KUKA KRL program: MyProgram_096().src

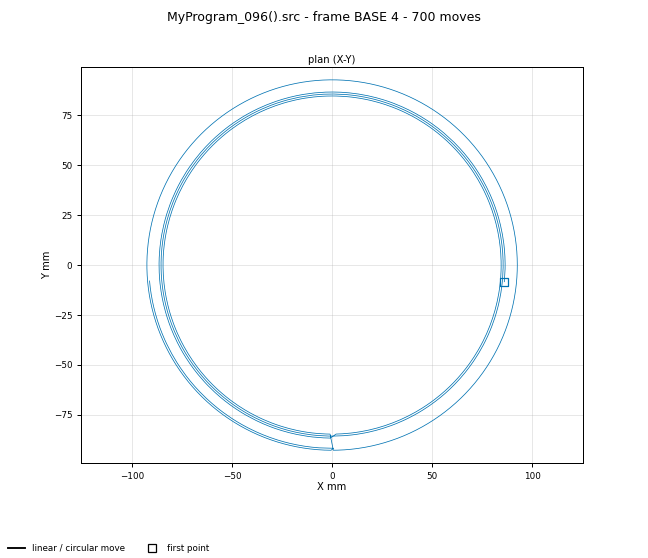
[picture p0: tool path of MyProgram_096().src in frame BASE 4, 700 of 700 moves have a stored position in this frame; points joined in program order, loops and branches not executed]
&ACCESS RVP
&REL 1
&PARAM TEMPLATE = C:\KRC\Roboter\Template\vorgabe
&PARAM EDITMASK = *
DEF MyProgram_096()
; ---- Setting reference (Base) ----
$BASE = BASE_DATA[4]

; --------------------------
; ---- Setting tool (TCP) ----
$TOOL = TOOL_DATA[3]
; --------------------------

$VEL.CP = VEL_APROX_PRINT
Startdeposition()
$VEL.CP = VEL_PRINT
LIN {X 86.1652,Y -8.3322,Z 89,A -10.037,B 24.913,C -2.1541,E1 25.1592,E2 454.8857} C_DIS
LIN {X 86.5449,Y -1.9567,Z 89,A -6.1016,B 24.9127,C -2.1574,E1 25.1598,E2 450.966} C_DIS
LIN {X 86.5649,Y 0.564,Z 89,A -3.5482,B 24.9097,C -2.1938,E1 25.1598,E2 448.3417} C_DIS
LIN {X 86.4537,Y 4.4277,Z 89,A -1.0805,B 24.9093,C -2.1987,E1 25.1594,E2 445.8771} C_DIS
LIN {X 86.1959,Y 7.9991,Z 89,A 0.4802,B 24.911,C -2.1778,E1 25.159,E2 444.3749} C_DIS
LIN {X 85.8962,Y 10.7562,Z 89,A 3.3475,B 24.9076,C -2.2199,E1 25.158,E2 441.4254} C_DIS
LIN {X 85.2355,Y 15.1219,Z 89,A 5.3712,B 24.9094,C -2.1974,E1 25.1571,E2 439.4666} C_DIS
LIN {X 84.2333,Y 19.9676,Z 89,A 8.7324,B 24.9083,C -2.2104,E1 25.1551,E2 436.0942} C_DIS
LIN {X 83.3839,Y 23.2585,Z 89,A 11.371,B 24.9066,C -2.2309,E1 25.1531,E2 433.4224} C_DIS
LIN {X 82.4594,Y 26.3489,Z 89,A 13.082,B 24.9073,C -2.2224,E1 25.1517,E2 431.7411} C_DIS
LIN {X 81.4082,Y 29.4361,Z 89,A 15.0667,B 24.9073,C -2.2228,E1 25.1499,E2 429.7667} C_DIS
LIN {X 80.3466,Y 32.2233,Z 89,A 17.2208,B 24.9063,C -2.2347,E1 25.1476,E2 427.5963} C_DIS
LIN {X 79.0048,Y 35.3836,Z 89,A 19.357,B 24.9062,C -2.2365,E1 25.1453,E2 425.4676} C_DIS
LIN {X 77.227,Y 39.1127,Z 89,A 22.0396,B 24.9057,C -2.2423,E1 25.142,E2 422.7857} C_DIS
LIN {X 75.0008,Y 43.2274,Z 89,A 24.8005,B 24.9059,C -2.2392,E1 25.1383,E2 420.0465} C_DIS
LIN {X 73.7426,Y 45.3426,Z 89,A 26.77,B 24.9046,C -2.2551,E1 25.1354,E2 418.0496} C_DIS
LIN {X 71.7448,Y 48.4398,Z 89,A 29.0057,B 24.9046,C -2.2544,E1 25.132,E2 415.8267} C_DIS
LIN {X 70.1596,Y 50.7113,Z 89,A 31.6144,B 24.902,C -2.2854,E1 25.1277,E2 413.1572} C_DIS
LIN {X 68.0698,Y 53.4816,Z 89,A 33.2305,B 24.9035,C -2.2677,E1 25.125,E2 411.5907} C_DIS
LIN {X 66.2061,Y 55.7736,Z 89,A 35.314,B 24.9028,C -2.2766,E1 25.1212,E2 409.4958} C_DIS
LIN {X 64.0318,Y 58.2561,Z 89,A 38.2857,B 24.9,C -2.3083,E1 25.1156,E2 406.4622} C_DIS
LIN {X 60.9971,Y 61.4257,Z 89,A 40.2743,B 24.9022,C -2.2834,E1 25.1118,E2 404.541} C_DIS
LIN {X 56.0568,Y 65.9649,Z 89,A 44.1821,B 24.9029,C -2.2744,E1 25.1038,E2 400.6702} C_DIS
LIN {X 53.2501,Y 68.2526,Z 89,A 47.0391,B 24.9013,C -2.2941,E1 25.0975,E2 397.7774} C_DIS
LIN {X 50.041,Y 70.6378,Z 89,A 49.6019,B 24.9011,C -2.2959,E1 25.0917,E2 395.2194} C_DIS
LIN {X 47.7464,Y 72.2081,Z 89,A 51.972,B 24.8993,C -2.3165,E1 25.0861,E2 392.8085} C_DIS
LIN {X 44.2677,Y 74.3919,Z 89,A 54.2125,B 24.9003,C -2.3047,E1 25.0809,E2 390.603} C_DIS
LIN {X 41.8224,Y 75.7944,Z 89,A 56.1926,B 24.8998,C -2.3111,E1 25.076,E2 388.6136} C_DIS
LIN {X 38.5837,Y 77.4922,Z 89,A 58.4027,B 24.9001,C -2.3073,E1 25.0706,E2 386.4186} C_DIS
LIN {X 34.9888,Y 79.1814,Z 89,A 61.2752,B 24.8992,C -2.3183,E1 25.0633,E2 383.5273} C_DIS
LIN {X 30.7564,Y 80.9183,Z 89,A 63.8229,B 24.9002,C -2.3058,E1 25.0568,E2 381.0151} C_DIS
LIN {X 28.2145,Y 81.8406,Z 89,A 65.9642,B 24.8991,C -2.3187,E1 25.051,E2 378.8475} C_DIS
LIN {X 25.6479,Y 82.6795,Z 89,A 67.7739,B 24.8989,C -2.3208,E1 25.0462,E2 377.0361} C_DIS
LIN {X 22.2469,Y 83.6595,Z 89,A 70.3552,B 24.8981,C -2.33,E1 25.0392,E2 374.4372} C_DIS
LIN {X 18.0288,Y 84.6691,Z 89,A 72.9776,B 24.8987,C -2.3235,E1 25.0321,E2 371.8337} C_DIS
LIN {X 13.1799,Y 85.557,Z 89,A 77.2175,B 24.8959,C -2.3559,E1 25.0203,E2 367.5214} C_DIS
LIN {X 8.4606,Y 86.1533,Z 89,A 79.4585,B 24.8984,C -2.3274,E1 25.0142,E2 365.3495} C_DIS
LIN {X 4.3743,Y 86.4555,Z 89,A 82.1881,B 24.8984,C -2.328,E1 25.0066,E2 362.6195} C_DIS
LIN {X 0.4649,Y 86.565,Z 89,A 84.9734,B 24.8978,C -2.3338,E1 24.9988,E2 359.821} C_DIS
LIN {X -3.1987,Y 86.5087,Z 89,A 88.381,B 24.8951,C -2.3638,E1 24.9891,E2 356.3412} C_DIS
LIN {X -8.7789,Y 86.1203,Z 89,A 90.702,B 24.8991,C -2.319,E1 24.9829,E2 354.1257} C_DIS
LIN {X -14.3867,Y 85.3625,Z 89,A 94.3706,B 24.8995,C -2.3142,E1 24.9728,E2 350.4655} C_DIS
LIN {X -17.7226,Y 84.7333,Z 89,A 97.0609,B 24.8985,C -2.3259,E1 24.9654,E2 347.7444} C_DIS
LIN {X -21.2707,Y 83.9126,Z 89,A 99.7429,B 24.898,C -2.3319,E1 24.958,E2 345.0444} C_DIS
LIN {X -24.8815,Y 82.9138,Z 89,A 101.8095,B 24.8993,C -2.3166,E1 24.9526,E2 343.0107} C_DIS
LIN {X -28.1429,Y 81.8655,Z 89,A 104.0096,B 24.8997,C -2.3119,E1 24.9468,E2 340.8178} C_DIS
LIN {X -32.7128,Y 80.1473,Z 89,A 107.0659,B 24.9005,C -2.3023,E1 24.9389,E2 337.7777} C_DIS
LIN {X -36.9162,Y 78.3013,Z 89,A 110.2494,B 24.9005,C -2.3021,E1 24.9307,E2 334.5871} C_DIS
LIN {X -39.8368,Y 76.8569,Z 89,A 112.4132,B 24.9009,C -2.2988,E1 24.9253,E2 332.4253} C_DIS
LIN {X -42.6915,Y 75.3087,Z 89,A 114.5747,B 24.9011,C -2.2955,E1 24.9201,E2 330.2655} C_DIS
LIN {X -44.87,Y 74.0298,Z 89,A 116.3495,B 24.9011,C -2.2955,E1 24.9158,E2 328.4852} C_DIS
LIN {X -49.0838,Y 71.3068,Z 89,A 119.6977,B 24.9016,C -2.2899,E1 24.908,E2 325.1394} C_DIS
LIN {X -51.7362,Y 69.406,Z 89,A 122.1888,B 24.9012,C -2.2952,E1 24.9024,E2 322.6269} C_DIS
LIN {X -54.4997,Y 67.257,Z 89,A 124.5303,B 24.9015,C -2.2909,E1 24.8973,E2 320.2868} C_DIS
LIN {X -58.1437,Y 64.135,Z 89,A 127.8803,B 24.9017,C -2.2888,E1 24.8903,E2 316.9286} C_DIS
LIN {X -60.4941,Y 61.9199,Z 89,A 129.6741,B 24.903,C -2.2737,E1 24.8867,E2 315.1632} C_DIS
LIN {X -63.2937,Y 59.0571,Z 89,A 132.285,B 24.9037,C -2.2661,E1 24.8817,E2 312.5592} C_DIS
LIN {X -65.8738,Y 56.1637,Z 89,A 135.6513,B 24.9022,C -2.2827,E1 24.8755,E2 309.1378} C_DIS
LIN {X -68.7539,Y 52.5995,Z 89,A 137.668,B 24.9054,C -2.2454,E1 24.8722,E2 307.2008} C_DIS
LIN {X -71.5133,Y 48.7816,Z 89,A 140.6821,B 24.9064,C -2.2339,E1 24.8673,E2 304.1992} C_DIS
LIN {X -72.8089,Y 46.825,Z 89,A 142.4997,B 24.9061,C -2.2371,E1 24.8645,E2 302.3648} C_DIS
LIN {X -75.3983,Y 42.5318,Z 89,A 145.8903,B 24.9067,C -2.2297,E1 24.8597,E2 298.9745} C_DIS
LIN {X -76.9384,Y 39.6775,Z 89,A 147.9529,B 24.9075,C -2.221,E1 24.857,E2 296.9215} C_DIS
LIN {X -78.2041,Y 37.1214,Z 89,A 149.991,B 24.9075,C -2.2197,E1 24.8545,E2 294.8756} C_DIS
LIN {X -80.0414,Y 32.9731,Z 89,A 152.6386,B 24.9092,C -2.2006,E1 24.8516,E2 292.2589} C_DIS
LIN {X -80.9706,Y 30.6182,Z 89,A 154.878,B 24.9083,C -2.2114,E1 24.8494,E2 289.9811} C_DIS
LIN {X -82.6055,Y 25.8867,Z 89,A 158.1523,B 24.9092,C -2.2001,E1 24.8465,E2 286.7152} C_DIS
LIN {X -83.441,Y 23.0556,Z 89,A 159.9044,B 24.9102,C -2.1882,E1 24.8452,E2 284.9813} C_DIS
LIN {X -84.156,Y 20.2864,Z 89,A 161.7857,B 24.9107,C -2.1819,E1 24.8439,E2 283.1039} C_DIS
LIN {X -85.1399,Y 15.6532,Z 89,A 165.0153,B 24.9113,C -2.1746,E1 24.8421,E2 279.8727} C_DIS
LIN {X -85.6777,Y 12.3726,Z 89,A 167.8753,B 24.9103,C -2.1863,E1 24.841,E2 276.9677} C_DIS
LIN {X -86.149,Y 8.5042,Z 89,A 169.6403,B 24.9129,C -2.155,E1 24.8405,E2 275.2669} C_DIS
LIN {X -86.4853,Y 3.7439,Z 89,A 172.8591,B 24.9136,C -2.1466,E1 24.8399,E2 272.0489} C_DIS
LIN {X -86.5642,Y 0.6968,Z 89,A 175.0036,B 24.9138,C -2.1437,E1 24.8398,E2 269.8984} C_DIS
LIN {X -86.4823,Y -3.8138,Z 89,A 178.5276,B 24.9133,C -2.1494,E1 24.8401,E2 266.3394} C_DIS
LIN {X -86.2728,Y -7.126,Z 89,A 179.9255,B 24.9157,C -2.1199,E1 24.8404,E2 265.0037} C_DIS
LIN {X -86.056,Y -9.3927,Z 89,A -177.5698,B 24.9138,C -2.1434,E1 24.8412,E2 262.4278} C_DIS
LIN {X -85.5563,Y -13.185,Z 89,A -175.8758,B 24.9164,C -2.1117,E1 24.8418,E2 260.7995} C_DIS
LIN {X -84.9399,Y -16.705,Z 89,A -173.2886,B 24.9164,C -2.1106,E1 24.8431,E2 258.1996} C_DIS
LIN {X -84.2882,Y -19.7303,Z 89,A -171.2652,B 24.917,C -2.1036,E1 24.8444,E2 256.1809} C_DIS
LIN {X -83.3415,Y -23.4082,Z 89,A -169.0394,B 24.9183,C -2.0878,E1 24.846,E2 253.9799} C_DIS
LIN {X -82.6319,Y -25.8014,Z 89,A -167.0637,B 24.9179,C -2.092,E1 24.8476,E2 251.9827} C_DIS
LIN {X -81.5331,Y -29.0907,Z 89,A -164.6138,B 24.9181,C -2.0897,E1 24.8498,E2 249.5246} C_DIS
LIN {X -80.5182,Y -31.7893,Z 89,A -162.9315,B 24.919,C -2.0777,E1 24.8515,E2 247.8614} C_DIS
LIN {X -79.1289,Y -35.1047,Z 89,A -160.0378,B 24.9184,C -2.0857,E1 24.8548,E2 244.9325} C_DIS
LIN {X -77.4475,Y -38.6738,Z 89,A -157.6886,B 24.9196,C -2.0709,E1 24.8576,E2 242.606} C_DIS
LIN {X -75.9339,Y -41.5677,Z 89,A -155.686,B 24.9204,C -2.0604,E1 24.8602,E2 240.6178} C_DIS
LIN {X -74.4678,Y -44.1393,Z 89,A -153.6152,B 24.9205,C -2.0585,E1 24.8632,E2 238.5409} C_DIS
LIN {X -73.1265,Y -46.3303,Z 89,A -152.1316,B 24.9214,C -2.0478,E1 24.8653,E2 237.0753} C_DIS
LIN {X -71.2162,Y -49.2139,Z 89,A -149.0869,B 24.9201,C -2.064,E1 24.8702,E2 233.9767} C_DIS
LIN {X -69.1788,Y -52.0385,Z 89,A -147.1357,B 24.9213,C -2.0481,E1 24.8734,E2 232.0542} C_DIS
LIN {X -67.1011,Y -54.692,Z 89,A -145.069,B 24.9221,C -2.038,E1 24.877,E2 230.0018} C_DIS
LIN {X -63.8641,Y -58.4389,Z 89,A -142.2392,B 24.9237,C -2.0175,E1 24.8822,E2 227.2081} C_DIS
LIN {X -62.2823,Y -60.1219,Z 89,A -140.3571,B 24.9231,C -2.0245,E1 24.8858,E2 225.3011} C_DIS
LIN {X -58.6037,Y -63.7129,Z 89,A -136.8514,B 24.9234,C -2.0206,E1 24.8929,E2 221.7902} C_DIS
LIN {X -56.0418,Y -65.9776,Z 89,A -134.6035,B 24.9238,C -2.0158,E1 24.8976,E2 219.5451} C_DIS
LIN {X -53.545,Y -68.0196,Z 89,A -132.3743,B 24.9238,C -2.0147,E1 24.9025,E2 217.3101} C_DIS
LIN {X -50.9969,Y -69.9504,Z 89,A -129.8993,B 24.9233,C -2.0219,E1 24.9081,E2 214.8092} C_DIS
LIN {X -48.1446,Y -71.9447,Z 89,A -127.8708,B 24.9243,C -2.0098,E1 24.9128,E2 212.8027} C_DIS
LIN {X -45.3206,Y -73.756,Z 89,A -125.9165,B 24.9251,C -1.9984,E1 24.9173,E2 210.8692} C_DIS
LIN {X -43.0007,Y -75.1311,Z 89,A -123.765,B 24.9245,C -2.007,E1 24.9226,E2 208.6908} C_DIS
LIN {X -37.8884,Y -77.8356,Z 89,A -120.3477,B 24.9258,C -1.9896,E1 24.931,E2 205.3056} C_DIS
LIN {X -34.2947,Y -79.4839,Z 89,A -117.631,B 24.9258,C -1.9898,E1 24.9379,E2 202.5819} C_DIS
LIN {X -31.1627,Y -80.7643,Z 89,A -115.3064,B 24.9258,C -1.9902,E1 24.944,E2 200.2512} C_DIS
LIN {X -28.6047,Y -81.7037,Z 89,A -113.5823,B 24.926,C -1.9862,E1 24.9485,E2 198.5332} C_DIS
LIN {X -25.2724,Y -82.7959,Z 89,A -110.8821,B 24.9253,C -1.9963,E1 24.9558,E2 195.8044} C_DIS
LIN {X -21.5951,Y -83.8294,Z 89,A -108.5996,B 24.926,C -1.9871,E1 24.9619,E2 193.5403} C_DIS
LIN {X -17.6457,Y -84.7486,Z 89,A -106.0736,B 24.9264,C -1.9809,E1 24.9687,E2 191.0258} C_DIS
LIN {X -12.0537,Y -85.723,Z 89,A -102.4921,B 24.9269,C -1.9741,E1 24.9786,E2 187.4568} C_DIS
LIN {X -9.5862,Y -86.0352,Z 89,A -100.3696,B 24.9258,C -1.9889,E1 24.9845,E2 185.2978} C_DIS
LIN {X -4.2582,Y -86.4608,Z 89,A -96.8864,B 24.926,C -1.9873,E1 24.9942,E2 181.8172} C_DIS
LIN {X -0.9571,Y -86.562,Z 89,A -94.6458,B 24.9258,C -1.9894,E1 25.0005,E2 179.5716} C_DIS
LIN {X -0.9571,Y -86.562,Z 89,A -94.6458,B 24.9258,C -1.9894,E1 25.0005,E2 179.5716} C_DIS
Enddeposition()
LIN {X 0.5384,Y -85.5676,Z 89,A -92.9762,B 24.9228,C -2.0285,E1 25.0055,E2 177.8093} C_DIS
Startdeposition()
$VEL.CP = VEL_PRINT
LIN {X -1.8149,Y -85.5541,Z 89,A -96.7949,B 24.9282,C -1.9573,E1 24.9943,E2 181.7968} C_DIS
LIN {X -7.3834,Y -85.2553,Z 89,A -99.9511,B 24.9269,C -1.975,E1 24.9856,E2 184.9121} C_DIS
LIN {X -10.1639,Y -84.9675,Z 89,A -101.8253,B 24.9269,C -1.9752,E1 24.9804,E2 186.787} C_DIS
LIN {X -14.2461,Y -84.379,Z 89,A -104.8301,B 24.9274,C -1.9684,E1 24.9721,E2 189.8105} C_DIS
LIN {X -18.2268,Y -83.6094,Z 89,A -107.4223,B 24.927,C -1.9733,E1 24.965,E2 192.3942} C_DIS
LIN {X -21.0814,Y -82.9359,Z 89,A -109.4344,B 24.927,C -1.9729,E1 24.9595,E2 194.41} C_DIS
LIN {X -23.2275,Y -82.3604,Z 89,A -110.8461,B 24.9268,C -1.9761,E1 24.9557,E2 195.8162} C_DIS
LIN {X -25.9725,Y -81.5373,Z 89,A -112.9249,B 24.927,C -1.9727,E1 24.9502,E2 197.9068} C_DIS
LIN {X -29.1962,Y -80.4385,Z 89,A -115.1571,B 24.9268,C -1.976,E1 24.9443,E2 200.1353} C_DIS
LIN {X -32.3957,Y -79.2041,Z 89,A -117.498,B 24.9268,C -1.9769,E1 24.9382,E2 202.4792} C_DIS
LIN {X -34.7519,Y -78.1996,Z 89,A -119.2917,B 24.9268,C -1.9764,E1 24.9336,E2 204.2784} C_DIS
LIN {X -38.4653,Y -76.4417,Z 89,A -121.9779,B 24.9264,C -1.9816,E1 24.9269,E2 206.9593} C_DIS
LIN {X -40.873,Y -75.1807,Z 89,A -123.6243,B 24.9258,C -1.9891,E1 24.9228,E2 208.5924} C_DIS
LIN {X -43.3867,Y -73.7589,Z 89,A -125.7047,B 24.9259,C -1.9875,E1 24.9178,E2 210.6828} C_DIS
LIN {X -46.2938,Y -71.9696,Z 89,A -128.0158,B 24.9257,C -1.9902,E1 24.9123,E2 212.9948} C_DIS
LIN {X -48.9738,Y -70.1736,Z 89,A -130.2026,B 24.9255,C -1.9929,E1 24.9073,E2 215.1825} C_DIS
LIN {X -51.5458,Y -68.3067,Z 89,A -132.2676,B 24.9251,C -1.9984,E1 24.9027,E2 217.2417} C_DIS
LIN {X -54.0811,Y -66.3178,Z 89,A -134.508,B 24.9251,C -1.9999,E1 24.8978,E2 219.4869} C_DIS
LIN {X -56.6656,Y -64.1249,Z 89,A -136.8256,B 24.9248,C -2.0029,E1 24.8929,E2 221.8065} C_DIS
LIN {X -58.5379,Y -62.4186,Z 89,A -138.4467,B 24.9244,C -2.0085,E1 24.8896,E2 223.4209} C_DIS
LIN {X -60.8702,Y -60.1462,Z 89,A -140.5817,B 24.9239,C -2.0143,E1 24.8853,E2 225.551} C_DIS
LIN {X -63.0112,Y -57.8994,Z 89,A -142.5919,B 24.9234,C -2.0208,E1 24.8815,E2 227.5546} C_DIS
LIN {X -64.8576,Y -55.8249,Z 89,A -144.6641,B 24.9236,C -2.0189,E1 24.8777,E2 229.6406} C_DIS
LIN {X -67.051,Y -53.1689,Z 89,A -146.7937,B 24.9228,C -2.0293,E1 24.8739,E2 231.7552} C_DIS
LIN {X -69.5729,Y -49.8234,Z 89,A -150.249,B 24.9236,C -2.018,E1 24.8682,E2 235.2544} C_DIS
LIN {X -71.3942,Y -47.1765,Z 89,A -151.5228,B 24.9214,C -2.048,E1 24.8663,E2 236.4629} C_DIS
LIN {X -73.247,Y -44.2456,Z 89,A -154.2983,B 24.9219,C -2.0412,E1 24.8621,E2 239.2686} C_DIS
LIN {X -74.9459,Y -41.3047,Z 89,A -156.6234,B 24.9215,C -2.0459,E1 24.8589,E2 241.5949} C_DIS
LIN {X -76.6041,Y -38.1389,Z 89,A -158.5908,B 24.9201,C -2.0643,E1 24.8565,E2 243.5288} C_DIS
LIN {X -78.9168,Y -33.0893,Z 89,A -162.522,B 24.9197,C -2.0688,E1 24.8519,E2 247.4707} C_DIS
LIN {X -80.3338,Y -29.4832,Z 89,A -165.2714,B 24.9195,C -2.0721,E1 24.8492,E2 250.2278} C_DIS
LIN {X -81.439,Y -26.2762,Z 89,A -167.6499,B 24.9192,C -2.0759,E1 24.8471,E2 252.611} C_DIS
LIN {X -82.4274,Y -22.991,Z 89,A -169.952,B 24.9187,C -2.0826,E1 24.8453,E2 254.9102} C_DIS
LIN {X -83.2905,Y -19.6361,Z 89,A -171.9622,B 24.9174,C -2.0982,E1 24.8439,E2 256.895} C_DIS
LIN {X -83.8501,Y -17.0858,Z 89,A -174.0038,B 24.9176,C -2.0955,E1 24.8427,E2 258.9549} C_DIS
LIN {X -84.4897,Y -13.5829,Z 89,A -176.2039,B 24.9167,C -2.1079,E1 24.8417,E2 261.1385} C_DIS
LIN {X -84.8798,Y -10.8714,Z 89,A -178.1199,B 24.9164,C -2.1115,E1 24.8409,E2 263.0575} C_DIS
LIN {X -85.2436,Y -7.5095,Z 89,A 179.5778,B 24.9159,C -2.1176,E1 24.8403,E2 265.359} C_DIS
LIN {X -85.4548,Y -4.5016,Z 89,A 177.5208,B 24.9155,C -2.1229,E1 24.8399,E2 267.4156} C_DIS
LIN {X -85.5573,Y -1.6423,Z 89,A 175.57,B 24.9151,C -2.1281,E1 24.8398,E2 269.3659} C_DIS
LIN {X -85.5639,Y 1.2851,Z 89,A 173.5749,B 24.9146,C -2.1334,E1 24.8398,E2 271.3603} C_DIS
LIN {X -85.4292,Y 4.965,Z 89,A 170.9832,B 24.9143,C -2.1379,E1 24.8402,E2 273.9569} C_DIS
LIN {X -85.1495,Y 8.5125,Z 89,A 168.4041,B 24.9141,C -2.1401,E1 24.8408,E2 276.546} C_DIS
LIN {X -84.6897,Y 12.2655,Z 89,A 166.2108,B 24.9127,C -2.1574,E1 24.8416,E2 278.7112} C_DIS
LIN {X -84.2353,Y 15.0718,Z 89,A 164.2791,B 24.9123,C -2.1627,E1 24.8425,E2 280.6417} C_DIS
LIN {X -83.8427,Y 17.1218,Z 89,A 162.8423,B 24.912,C -2.1661,E1 24.8433,E2 282.079} C_DIS
LIN {X -83.1416,Y 20.2539,Z 89,A 160.6118,B 24.9116,C -2.1706,E1 24.8447,E2 284.3117} C_DIS
LIN {X -82.4713,Y 22.836,Z 89,A 158.6992,B 24.9115,C -2.1728,E1 24.8461,E2 286.2304} C_DIS
LIN {X -81.0975,Y 27.312,Z 89,A 155.2618,B 24.9113,C -2.1743,E1 24.8491,E2 289.6837} C_DIS
LIN {X -79.516,Y 31.624,Z 89,A 152.7849,B 24.9092,C -2.2,E1 24.8515,E2 292.1133} C_DIS
LIN {X -78.1565,Y 34.8486,Z 89,A 150.2383,B 24.9091,C -2.2015,E1 24.8543,E2 294.6704} C_DIS
LIN {X -76.7924,Y 37.7591,Z 89,A 148.0261,B 24.9087,C -2.2062,E1 24.857,E2 296.8833} C_DIS
LIN {X -75.1867,Y 40.8621,Z 89,A 145.9149,B 24.9076,C -2.2193,E1 24.8597,E2 298.9745} C_DIS
LIN {X -73.913,Y 43.1253,Z 89,A 143.8292,B 24.908,C -2.2148,E1 24.8626,E2 301.0819} C_DIS
LIN {X -72.0009,Y 46.2451,Z 89,A 141.56,B 24.907,C -2.2266,E1 24.866,E2 303.3343} C_DIS
LIN {X -70.3404,Y 48.7339,Z 89,A 139.446,B 24.9068,C -2.2291,E1 24.8693,E2 305.4529} C_DIS
LIN {X -67.4202,Y 52.7017,Z 89,A 136.1098,B 24.9061,C -2.2369,E1 24.8749,E2 308.7866} C_DIS
LIN {X -65.4151,Y 55.1705,Z 89,A 134.0426,B 24.9055,C -2.2441,E1 24.8785,E2 310.8462} C_DIS
LIN {X -62.6012,Y 58.343,Z 89,A 130.9167,B 24.9055,C -2.2433,E1 24.8844,E2 313.9879} C_DIS
LIN {X -59.6674,Y 61.3408,Z 89,A 128.2728,B 24.9046,C -2.2545,E1 24.8896,E2 316.6161} C_DIS
LIN {X -57.164,Y 63.6792,Z 89,A 125.6556,B 24.905,C -2.2508,E1 24.8951,E2 319.2528} C_DIS
LIN {X -53.5029,Y 66.7864,Z 89,A 122.6793,B 24.9038,C -2.2645,E1 24.9014,E2 322.2077} C_DIS
LIN {X -50.968,Y 68.7406,Z 89,A 120.6628,B 24.9031,C -2.2725,E1 24.9059,E2 324.2124} C_DIS
LIN {X -48.7449,Y 70.3327,Z 89,A 118.9125,B 24.9026,C -2.2785,E1 24.9099,E2 325.9544} C_DIS
LIN {X -46.2633,Y 71.9892,Z 89,A 116.7706,B 24.9026,C -2.2782,E1 24.9149,E2 328.104} C_DIS
LIN {X -43.3634,Y 73.7726,Z 89,A 114.4744,B 24.9023,C -2.2819,E1 24.9204,E2 330.3985} C_DIS
LIN {X -40.4184,Y 75.4274,Z 89,A 112.1744,B 24.9021,C -2.2846,E1 24.926,E2 332.6986} C_DIS
LIN {X -37.4397,Y 76.9493,Z 89,A 109.9397,B 24.9018,C -2.2883,E1 24.9316,E2 334.9303} C_DIS
LIN {X -35.0528,Y 78.0645,Z 89,A 108.0014,B 24.902,C -2.286,E1 24.9366,E2 336.879} C_DIS
LIN {X -30.8751,Y 79.8102,Z 89,A 105.1011,B 24.9013,C -2.2939,E1 24.944,E2 339.7668} C_DIS
LIN {X -27.778,Y 80.9403,Z 89,A 102.9222,B 24.901,C -2.2975,E1 24.9497,E2 341.9415} C_DIS
LIN {X -24.5146,Y 81.9867,Z 89,A 101.0452,B 24.8997,C -2.3124,E1 24.9547,E2 343.7864} C_DIS
LIN {X -22.3942,Y 82.5909,Z 89,A 98.806,B 24.9015,C -2.2916,E1 24.9608,E2 346.0786} C_DIS
LIN {X -16.6055,Y 83.9475,Z 89,A 95.1889,B 24.9003,C -2.3057,E1 24.9706,E2 349.6665} C_DIS
LIN {X -9.4624,Y 85.0497,Z 89,A 90.5621,B 24.8994,C -2.3152,E1 24.9834,E2 354.2746} C_DIS
LIN {X -4.2831,Y 85.4669,Z 89,A 86.8264,B 24.9,C -2.309,E1 24.9938,E2 358.0266} C_DIS
LIN {X 0.7813,Y 85.5698,Z 89,A 83.5768,B 24.8995,C -2.3141,E1 25.0028,E2 361.2643} C_DIS
LIN {X 7.2171,Y 85.2691,Z 89,A 79.1927,B 24.8997,C -2.312,E1 25.0151,E2 365.6517} C_DIS
LIN {X 10.7912,Y 84.8901,Z 89,A 76.7737,B 24.8997,C -2.3112,E1 25.0218,E2 368.0708} C_DIS
LIN {X 13.3554,Y 84.5249,Z 89,A 74.9622,B 24.9,C -2.3083,E1 25.0268,E2 369.8874} C_DIS
LIN {X 16.5222,Y 83.9636,Z 89,A 72.872,B 24.9,C -2.3094,E1 25.0325,E2 371.9727} C_DIS
LIN {X 19.5039,Y 83.3211,Z 89,A 71.0544,B 24.8994,C -2.3154,E1 25.0374,E2 373.7738} C_DIS
LIN {X 21.4099,Y 82.8515,Z 89,A 69.5187,B 24.9001,C -2.3077,E1 25.0416,E2 375.3253} C_DIS
LIN {X 23.8106,Y 82.1952,Z 89,A 67.7064,B 24.9006,C -2.302,E1 25.0465,E2 377.1481} C_DIS
LIN {X 27.0631,Y 81.1814,Z 89,A 65.8618,B 24.8995,C -2.3139,E1 25.0513,E2 378.9612} C_DIS
LIN {X 29.4806,Y 80.3347,Z 89,A 63.8265,B 24.9006,C -2.3023,E1 25.0568,E2 381.0197} C_DIS
LIN {X 32.3928,Y 79.2052,Z 89,A 61.7398,B 24.9007,C -2.3003,E1 25.0622,E2 383.1064} C_DIS
LIN {X 36.5342,Y 77.3835,Z 89,A 58.6973,B 24.9011,C -2.2965,E1 25.0699,E2 386.1505} C_DIS
LIN {X 39.243,Y 76.045,Z 89,A 56.6895,B 24.9012,C -2.2944,E1 25.0749,E2 388.1577} C_DIS
LIN {X 42.1741,Y 74.4604,Z 89,A 54.4389,B 24.9016,C -2.2907,E1 25.0804,E2 390.4105} C_DIS
LIN {X 45.0291,Y 72.7685,Z 89,A 52.5625,B 24.9009,C -2.2985,E1 25.0848,E2 392.2625} C_DIS
LIN {X 47.5447,Y 71.1514,Z 89,A 50.2165,B 24.9021,C -2.2842,E1 25.0904,E2 394.6345} C_DIS
LIN {X 50.4115,Y 69.148,Z 89,A 47.9492,B 24.9022,C -2.2827,E1 25.0955,E2 396.8976} C_DIS
LIN {X 53.0771,Y 67.1235,Z 89,A 45.7734,B 24.9024,C -2.2808,E1 25.1003,E2 399.07} C_DIS
LIN {X 55.8459,Y 64.8398,Z 89,A 42.9035,B 24.9041,C -2.2611,E1 25.1065,E2 401.9754} C_DIS
LIN {X 59.155,Y 61.8347,Z 89,A 40.3518,B 24.9034,C -2.2693,E1 25.1117,E2 404.4971} C_DIS
LIN {X 60.945,Y 60.0705,Z 89,A 38.3897,B 24.9045,C -2.2566,E1 25.1156,E2 406.4809} C_DIS
LIN {X 64.0701,Y 56.7273,Z 89,A 35.5601,B 24.9044,C -2.2575,E1 25.1209,E2 409.296} C_DIS
LIN {X 66.1353,Y 54.3057,Z 89,A 33.468,B 24.9047,C -2.2538,E1 25.1246,E2 411.3872} C_DIS
LIN {X 68.0726,Y 51.8564,Z 89,A 31.2683,B 24.9054,C -2.2452,E1 25.1284,E2 413.5968} C_DIS
LIN {X 70.3042,Y 48.786,Z 89,A 28.8801,B 24.9055,C -2.244,E1 25.1322,E2 415.9763} C_DIS
LIN {X 72.1626,Y 45.9933,Z 89,A 26.6439,B 24.906,C -2.2385,E1 25.1357,E2 418.2142} C_DIS
LIN {X 73.8847,Y 43.1738,Z 89,A 24.6595,B 24.9059,C -2.2403,E1 25.1385,E2 420.1844} C_DIS
LIN {X 75.5699,Y 40.1501,Z 89,A 22.1257,B 24.907,C -2.2268,E1 25.1419,E2 422.7368} C_DIS
LIN {X 77.2885,Y 36.7337,Z 89,A 19.5482,B 24.9076,C -2.2191,E1 25.1451,E2 425.3186} C_DIS
LIN {X 78.6528,Y 33.7157,Z 89,A 17.3383,B 24.9081,C -2.213,E1 25.1476,E2 427.5308} C_DIS
LIN {X 79.9336,Y 30.5521,Z 89,A 15.1318,B 24.9085,C -2.2091,E1 25.1498,E2 429.7344} C_DIS
LIN {X 81.0747,Y 27.3796,Z 89,A 13.0986,B 24.9084,C -2.21,E1 25.1517,E2 431.754} C_DIS
LIN {X 81.8882,Y 24.8462,Z 89,A 10.9794,B 24.9098,C -2.1932,E1 25.1535,E2 433.9007} C_DIS
LIN {X 82.8474,Y 21.4258,Z 89,A 8.8283,B 24.9098,C -2.1937,E1 25.155,E2 436.0383} C_DIS
LIN {X 83.5305,Y 18.5883,Z 89,A 6.3758,B 24.9116,C -2.1709,E1 25.1566,E2 438.5304} C_DIS
LIN {X 84.3922,Y 14.1668,Z 89,A 3.9931,B 24.9106,C -2.1829,E1 25.1577,E2 440.8707} C_DIS
LIN {X 85.0142,Y 9.7658,Z 89,A 1.0167,B 24.9114,C -2.1736,E1 25.1589,E2 443.8517} C_DIS
LIN {X 85.3494,Y 6.1873,Z 89,A -1.5916,B 24.9126,C -2.1591,E1 25.1595,E2 446.4788} C_DIS
LIN {X 85.5447,Y 2.1875,Z 89,A -4.5673,B 24.9141,C -2.1405,E1 25.1598,E2 449.4805} C_DIS
LIN {X 85.5644,Y -1.2567,Z 89,A -7.6995,B 24.9169,C -2.1054,E1 25.1596,E2 452.677} C_DIS
LIN {X 85.3008,Y -6.8205,Z 89,A -9.9181,B 24.9138,C -2.1444,E1 25.1592,E2 454.7903} C_DIS
LIN {X 85.0336,Y -9.5997,Z 89,A -12.4197,B 24.916,C -2.1169,E1 25.1585,E2 457.342} C_DIS
LIN {X 84.4544,Y -13.7951,Z 89,A -15.2211,B 24.9166,C -2.109,E1 25.1573,E2 460.1456} C_DIS
LIN {X 83.6557,Y -18.0145,Z 89,A -17.6207,B 24.916,C -2.116,E1 25.156,E2 462.5147} C_DIS
LIN {X 83.0449,Y -20.6503,Z 89,A -19.6154,B 24.917,C -2.104,E1 25.1546,E2 464.5261} C_DIS
LIN {X 82.119,Y -24.0686,Z 89,A -21.7992,B 24.917,C -2.103,E1 25.153,E2 466.6998} C_DIS
LIN {X 81.3189,Y -26.6473,Z 89,A -24.0082,B 24.9186,C -2.0837,E1 25.1511,E2 468.9418} C_DIS
LIN {X 79.8497,Y -30.7736,Z 89,A -26.385,B 24.9178,C -2.0936,E1 25.1488,E2 471.2822} C_DIS
LIN {X 78.9903,Y -32.915,Z 89,A -28.0874,B 24.9186,C -2.0835,E1 25.147,E2 472.9988} C_DIS
LIN {X 77.8564,Y -35.5145,Z 89,A -29.9288,B 24.9189,C -2.0797,E1 25.1449,E2 474.8392} C_DIS
LIN {X 76.6379,Y -38.0707,Z 89,A -31.7673,B 24.9192,C -2.0761,E1 25.1427,E2 476.6765} C_DIS
LIN {X 75.6533,Y -39.9918,Z 89,A -33.5836,B 24.9205,C -2.0593,E1 25.1403,E2 478.5228} C_DIS
LIN {X 73.4131,Y -43.9716,Z 89,A -36.8077,B 24.9216,C -2.0449,E1 25.1357,E2 481.7643} C_DIS
LIN {X 70.733,Y -48.1626,Z 89,A -39.3815,B 24.9203,C -2.0611,E1 25.1318,E2 484.287} C_DIS
LIN {X 68.3566,Y -51.4794,Z 89,A -42.2794,B 24.9213,C -2.048,E1 25.1271,E2 487.2017} C_DIS
LIN {X 66.5156,Y -53.837,Z 89,A -44.2858,B 24.9218,C -2.0426,E1 25.1236,E2 489.2115} C_DIS
LIN {X 64.0945,Y -56.7,Z 89,A -47.0956,B 24.923,C -2.0261,E1 25.1184,E2 492.0477} C_DIS
LIN {X 61.4088,Y -59.5969,Z 89,A -49.5195,B 24.923,C -2.0269,E1 25.1137,E2 494.459} C_DIS
LIN {X 59.0247,Y -61.9603,Z 89,A -51.5456,B 24.9228,C -2.0289,E1 25.1097,E2 496.472} C_DIS
LIN {X 56.6825,Y -64.1101,Z 89,A -54.1022,B 24.9243,C -2.0098,E1 25.1043,E2 499.0635} C_DIS
LIN {X 54.328,Y -66.1168,Z 89,A -56.3973,B 24.9252,C -1.9978,E1 25.0994,E2 501.3782} C_DIS
LIN {X 51.8004,Y -68.1154,Z 89,A -58.7307,B 24.9259,C -1.9875,E1 25.0941,E2 503.7275} C_DIS
LIN {X 48.7697,Y -70.3155,Z 89,A -60.5452,B 24.9246,C -2.0051,E1 25.0901,E2 505.494} C_DIS
LIN {X 45.5802,Y -72.4242,Z 89,A -62.9726,B 24.9246,C -2.0045,E1 25.0844,E2 507.9148} C_DIS
LIN {X 43.3427,Y -73.7849,Z 89,A -64.6957,B 24.9248,C -2.0023,E1 25.0803,E2 509.6378} C_DIS
LIN {X 41.0758,Y -75.0708,Z 89,A -66.6345,B 24.9255,C -1.9929,E1 25.0755,E2 511.5932} C_DIS
LIN {X 37.9914,Y -76.6772,Z 89,A -68.7978,B 24.9255,C -1.9944,E1 25.0702,E2 513.747} C_DIS
LIN {X 35.5461,Y -77.8422,Z 89,A -70.7811,B 24.926,C -1.9861,E1 25.0651,E2 515.745} C_DIS
LIN {X 32.3428,Y -79.2256,Z 89,A -73.0497,B 24.9261,C -1.9849,E1 25.0593,E2 518.0111} C_DIS
LIN {X 29.7634,Y -80.2313,Z 89,A -75.2888,B 24.9272,C -1.97,E1 25.0533,E2 520.2807} C_DIS
LIN {X 25.5848,Y -81.6592,Z 89,A -77.9069,B 24.9267,C -1.9772,E1 25.0465,E2 522.8766} C_DIS
LIN {X 21.8299,Y -82.7433,Z 89,A -80.5785,B 24.927,C -1.9727,E1 25.0392,E2 525.5548} C_DIS
LIN {X 18.6323,Y -83.5209,Z 89,A -82.7437,B 24.9271,C -1.9718,E1 25.0334,E2 527.719} C_DIS
LIN {X 16.3676,Y -83.9933,Z 89,A -84.8791,B 24.9286,C -1.952,E1 25.0274,E2 529.8987} C_DIS
LIN {X 12.5359,Y -84.6513,Z 89,A -86.8273,B 24.9272,C -1.9707,E1 25.0221,E2 531.8009} C_DIS
LIN {X 9.459,Y -85.0496,Z 89,A -88.9293,B 24.9273,C -1.9687,E1 25.0163,E2 533.9061} C_DIS
LIN {X 5.8623,Y -85.372,Z 89,A -90.9653,B 24.9265,C -1.9795,E1 25.0107,E2 535.9153} C_DIS
LIN {X 0.5384,Y -85.5676,Z 89,A -92.9744,B 24.9229,C -2.0277,E1 25.0055,E2 537.8093} C_DIS
Enddeposition()
LIN {X 0.5384,Y -85.5676,Z 89,A -92.9744,B 24.9229,C -2.0277,E1 25.0055,E2 537.8093} C_DIS
Startdeposition()
$VEL.CP = VEL_PRINT
LIN {X 1.9976,Y -84.5574,Z 89,A -92.9051,B 24.9238,C -2.0156,E1 25.0055,E2 537.7687} C_DIS
LIN {X 4.9247,Y -84.4367,Z 89,A -91.0545,B 24.9241,C -2.0122,E1 25.0107,E2 535.9269} C_DIS
LIN {X 7.2381,Y -84.271,Z 89,A -89.505,B 24.9241,C -2.0122,E1 25.015,E2 534.3781} C_DIS
LIN {X 9.3008,Y -84.0683,Z 89,A -88.1028,B 24.9241,C -2.013,E1 25.0189,E2 532.975} C_DIS
LIN {X 11.3852,Y -83.8116,Z 89,A -86.4291,B 24.9233,C -2.0219,E1 25.0236,E2 531.2816} C_DIS
LIN {X 14.475,Y -83.3335,Z 89,A -84.5624,B 24.9238,C -2.0155,E1 25.0287,E2 529.432} C_DIS
LIN {X 16.5066,Y -82.955,Z 89,A -83.1643,B 24.9238,C -2.0166,E1 25.0325,E2 528.033} C_DIS
LIN {X 18.5295,Y -82.5268,Z 89,A -81.7678,B 24.9237,C -2.0177,E1 25.0363,E2 526.6356} C_DIS
LIN {X 20.5418,Y -82.049,Z 89,A -80.3743,B 24.9236,C -2.0189,E1 25.0401,E2 525.2414} C_DIS
LIN {X 22.5422,Y -81.5221,Z 89,A -78.9763,B 24.9235,C -2.0202,E1 25.0439,E2 523.8424} C_DIS
LIN {X 24.5289,Y -80.9464,Z 89,A -77.5784,B 24.9234,C -2.0217,E1 25.0476,E2 522.4434} C_DIS
LIN {X 26.5137,Y -80.3182,Z 89,A -76.1721,B 24.9232,C -2.0233,E1 25.0513,E2 521.0361} C_DIS
LIN {X 28.4551,Y -79.651,Z 89,A -74.7852,B 24.9232,C -2.0249,E1 25.055,E2 519.648} C_DIS
LIN {X 30.3909,Y -78.9326,Z 89,A -73.389,B 24.923,C -2.0268,E1 25.0587,E2 518.2505} C_DIS
LIN {X 32.364,Y -78.1446,Z 89,A -71.9559,B 24.9228,C -2.0286,E1 25.0624,E2 516.8163} C_DIS
LIN {X 34.237,Y -77.3421,Z 89,A -70.5716,B 24.9227,C -2.0308,E1 25.0659,E2 515.4302} C_DIS
LIN {X 36.1708,Y -76.457,Z 89,A -69.1494,B 24.9225,C -2.0324,E1 25.0695,E2 514.0078} C_DIS
LIN {X 38.0302,Y -75.5494,Z 89,A -67.7489,B 24.9224,C -2.0347,E1 25.073,E2 512.6057} C_DIS
LIN {X 39.8545,Y -74.603,Z 89,A -66.3605,B 24.9222,C -2.0369,E1 25.0765,E2 511.2159} C_DIS
LIN {X 41.6673,Y -73.6059,Z 89,A -64.9643,B 24.922,C -2.0392,E1 25.0799,E2 509.8183} C_DIS
LIN {X 43.4667,Y -72.5579,Z 89,A -63.5599,B 24.9218,C -2.0416,E1 25.0832,E2 508.4127} C_DIS
LIN {X 45.2151,Y -71.4812,Z 89,A -62.1743,B 24.9217,C -2.044,E1 25.0865,E2 507.0257} C_DIS
LIN {X 47.4263,Y -70.032,Z 89,A -60.2925,B 24.9212,C -2.0506,E1 25.0909,E2 505.1346} C_DIS
LIN {X 49.4036,Y -68.6524,Z 89,A -58.7582,B 24.9212,C -2.0506,E1 25.0944,E2 503.6056} C_DIS
LIN {X 51.4999,Y -67.0934,Z 89,A -56.8088,B 24.9204,C -2.0603,E1 25.0988,E2 501.6404} C_DIS
LIN {X 54.4435,Y -64.7295,Z 89,A -54.4585,B 24.9204,C -2.059,E1 25.1038,E2 499.302} C_DIS
LIN {X 56.4142,Y -63.0173,Z 89,A -52.5881,B 24.9199,C -2.0665,E1 25.1078,E2 497.4213} C_DIS
LIN {X 58.6939,Y -60.8997,Z 89,A -50.4934,B 24.9196,C -2.071,E1 25.112,E2 495.3246} C_DIS
LIN {X 60.8942,Y -58.6996,Z 89,A -48.3976,B 24.9192,C -2.0758,E1 25.1161,E2 493.2265} C_DIS
LIN {X 63.007,Y -56.4258,Z 89,A -46.3016,B 24.9188,C -2.0808,E1 25.1201,E2 491.1278} C_DIS
LIN {X 65.0544,Y -54.0524,Z 89,A -44.1969,B 24.9184,C -2.0857,E1 25.1239,E2 489.0212} C_DIS
LIN {X 66.9954,Y -51.6272,Z 89,A -42.1025,B 24.918,C -2.091,E1 25.1275,E2 486.9242} C_DIS
LIN {X 68.5729,Y -49.515,Z 89,A -40.4545,B 24.918,C -2.0911,E1 25.1302,E2 485.2838} C_DIS
LIN {X 69.7484,Y -47.8452,Z 89,A -39.0642,B 24.9177,C -2.0952,E1 25.1324,E2 483.8907} C_DIS
LIN {X 70.8837,Y -46.1464,Z 89,A -37.6853,B 24.9174,C -2.0989,E1 25.1346,E2 482.51} C_DIS
LIN {X 71.9745,Y -44.4255,Z 89,A -36.3141,B 24.9171,C -2.1025,E1 25.1366,E2 481.1372} C_DIS
LIN {X 73.006,Y -42.7085,Z 89,A -34.968,B 24.9168,C -2.106,E1 25.1385,E2 479.7897} C_DIS
LIN {X 74.3828,Y -40.261,Z 89,A -32.9912,B 24.9162,C -2.1141,E1 25.1412,E2 477.8041} C_DIS
LIN {X 75.549,Y -38.031,Z 89,A -31.3807,B 24.916,C -2.1159,E1 25.1433,E2 476.1979} C_DIS
LIN {X 76.4569,Y -36.1712,Z 89,A -29.9879,B 24.9157,C -2.1198,E1 25.1449,E2 474.8034} C_DIS
LIN {X 77.313,Y -34.3027,Z 89,A -28.6046,B 24.9154,C -2.1236,E1 25.1465,E2 473.4185} C_DIS
LIN {X 78.1341,Y -32.389,Z 89,A -27.2037,B 24.9151,C -2.1276,E1 25.148,E2 472.016} C_DIS
LIN {X 78.9089,Y -30.4531,Z 89,A -25.8005,B 24.9148,C -2.1316,E1 25.1495,E2 470.611} C_DIS
LIN {X 79.6309,Y -28.5116,Z 89,A -24.4092,B 24.9145,C -2.1355,E1 25.1508,E2 469.2183} C_DIS
LIN {X 80.3128,Y -26.5306,Z 89,A -22.9978,B 24.9141,C -2.1397,E1 25.1521,E2 467.8052} C_DIS
LIN {X 80.9376,Y -24.5584,Z 89,A -21.6028,B 24.9138,C -2.1438,E1 25.1532,E2 466.4082} C_DIS
LIN {X 81.5141,Y -22.5712,Z 89,A -20.2132,B 24.9135,C -2.1478,E1 25.1543,E2 465.0172} C_DIS
LIN {X 82.0418,Y -20.5703,Z 89,A -18.8213,B 24.9131,C -2.1519,E1 25.1553,E2 463.6237} C_DIS
LIN {X 82.5204,Y -18.5573,Z 89,A -17.4295,B 24.9128,C -2.156,E1 25.1561,E2 462.2302} C_DIS
LIN {X 82.9495,Y -16.5337,Z 89,A -16.0376,B 24.9125,C -2.1601,E1 25.1569,E2 460.8367} C_DIS
LIN {X 83.3288,Y -14.5013,Z 89,A -14.647,B 24.9121,C -2.1643,E1 25.1576,E2 459.4445} C_DIS
LIN {X 83.6529,Y -12.495,Z 89,A -13.0248,B 24.9111,C -2.1771,E1 25.1583,E2 457.8017} C_DIS
LIN {X 84.1028,Y -8.9721,Z 89,A -10.7123,B 24.9107,C -2.1816,E1 25.159,E2 455.4922} C_DIS
LIN {X 84.3444,Y -6.3205,Z 89,A -8.9424,B 24.9104,C -2.1862,E1 25.1594,E2 453.7218} C_DIS
LIN {X 84.5254,Y -3.0696,Z 89,A -6.9312,B 24.9104,C -2.1866,E1 25.1597,E2 451.7216} C_DIS
LIN {X 84.5761,Y -0.9041,Z 89,A -5.2186,B 24.9092,C -2.1997,E1 25.1597,E2 449.9883} C_DIS
LIN {X 84.5573,Y 2.001,Z 89,A -3.4991,B 24.9094,C -2.1975,E1 25.1597,E2 448.2842} C_DIS
LIN {X 84.4855,Y 4.0101,Z 89,A -2.1512,B 24.9091,C -2.2014,E1 25.1596,E2 446.9351} C_DIS
LIN {X 84.3709,Y 5.9458,Z 89,A -0.8231,B 24.9087,C -2.206,E1 25.1593,E2 445.6039} C_DIS
LIN {X 84.1013,Y 8.9855,Z 89,A 1.2563,B 24.9081,C -2.213,E1 25.1588,E2 443.5204} C_DIS
LIN {X 83.6635,Y 12.4263,Z 89,A 3.5406,B 24.9077,C -2.2181,E1 25.1579,E2 441.2375} C_DIS
LIN {X 83.3381,Y 14.4487,Z 89,A 4.923,B 24.9074,C -2.2223,E1 25.1573,E2 439.8534} C_DIS
LIN {X 82.9609,Y 16.4765,Z 89,A 6.3108,B 24.907,C -2.2263,E1 25.1565,E2 438.4642} C_DIS
LIN {X 82.5708,Y 18.3275,Z 89,A 7.6069,B 24.9066,C -2.2308,E1 25.1558,E2 437.1651} C_DIS
LIN {X 82.0501,Y 20.5373,Z 89,A 9.3474,B 24.9057,C -2.2423,E1 25.1546,E2 435.4074} C_DIS
LIN {X 81.2373,Y 23.5479,Z 89,A 11.2096,B 24.9059,C -2.2402,E1 25.1532,E2 433.5608} C_DIS
LIN {X 80.6369,Y 25.5281,Z 89,A 12.602,B 24.9055,C -2.2441,E1 25.152,E2 432.1672} C_DIS
LIN {X 79.9797,Y 27.5184,Z 89,A 14.0106,B 24.9052,C -2.2479,E1 25.1508,E2 430.7575} C_DIS
LIN {X 79.2816,Y 29.4693,Z 89,A 15.4072,B 24.9049,C -2.2518,E1 25.1495,E2 429.3595} C_DIS
LIN {X 78.5359,Y 31.4025,Z 89,A 16.802,B 24.9046,C -2.2556,E1 25.148,E2 427.9636} C_DIS
LIN {X 77.4796,Y 33.9216,Z 89,A 18.708,B 24.9039,C -2.2628,E1 25.1459,E2 426.051} C_DIS
LIN {X 76.1935,Y 36.7192,Z 89,A 20.7933,B 24.9034,C -2.2686,E1 25.1435,E2 423.9633} C_DIS
LIN {X 75.0847,Y 38.9394,Z 89,A 22.3849,B 24.9034,C -2.2702,E1 25.1414,E2 422.3763} C_DIS
LIN {X 74.1065,Y 40.7704,Z 89,A 23.7826,B 24.903,C -2.2737,E1 25.1396,E2 420.9776} C_DIS
LIN {X 73.0756,Y 42.5908,Z 89,A 25.1908,B 24.9027,C -2.2772,E1 25.1376,E2 419.5685} C_DIS
LIN {X 72.0178,Y 44.3558,Z 89,A 26.5775,B 24.9024,C -2.2806,E1 25.1356,E2 418.1807} C_DIS
LIN {X 70.9024,Y 46.1179,Z 89,A 27.9822,B 24.9021,C -2.284,E1 25.1335,E2 416.7751} C_DIS
LIN {X 69.4961,Y 48.2084,Z 89,A 29.8182,B 24.9014,C -2.2927,E1 25.1306,E2 414.9277} C_DIS
LIN {X 67.936,Y 50.3856,Z 89,A 31.7014,B 24.9008,C -2.2994,E1 25.1275,E2 413.0377} C_DIS
LIN {X 66.0318,Y 52.8565,Z 89,A 33.8009,B 24.9004,C -2.304,E1 25.1238,E2 410.9372} C_DIS
LIN {X 64.0509,Y 55.2403,Z 89,A 35.892,B 24.9,C -2.3085,E1 25.12,E2 408.8449} C_DIS
LIN {X 61.9792,Y 57.555,Z 89,A 37.983,B 24.8996,C -2.3128,E1 25.1161,E2 406.7531} C_DIS
LIN {X 59.8108,Y 59.8053,Z 89,A 40.0933,B 24.8993,C -2.3171,E1 25.112,E2 404.6416} C_DIS
LIN {X 57.5779,Y 61.9579,Z 89,A 42.1829,B 24.8989,C -2.321,E1 25.1077,E2 402.5513} C_DIS
LIN {X 55.2482,Y 64.0441,Z 89,A 44.2952,B 24.8986,C -2.3249,E1 25.1033,E2 400.438} C_DIS
LIN {X 52.8591,Y 66.0297,Z 89,A 46.3898,B 24.8983,C -2.3285,E1 25.0987,E2 398.3429} C_DIS
LIN {X 50.3933,Y 67.9303,Z 89,A 48.2738,B 24.8986,C -2.325,E1 25.0946,E2 396.4742} C_DIS
LIN {X 48.7268,Y 69.1353,Z 89,A 49.8563,B 24.8978,C -2.3334,E1 25.0909,E2 394.8771} C_DIS
LIN {X 46.127,Y 70.8965,Z 89,A 51.7814,B 24.8981,C -2.3303,E1 25.0865,E2 392.9658} C_DIS
LIN {X 44.365,Y 72.0122,Z 89,A 53.1882,B 24.8979,C -2.3323,E1 25.0832,E2 391.5588} C_DIS
LIN {X 42.6001,Y 73.0701,Z 89,A 54.579,B 24.8978,C -2.3342,E1 25.0798,E2 390.1677} C_DIS
LIN {X 40.3452,Y 74.3371,Z 89,A 56.4408,B 24.8972,C -2.3402,E1 25.0753,E2 388.2973} C_DIS
LIN {X 37.5952,Y 75.7651,Z 89,A 58.5395,B 24.897,C -2.3428,E1 25.07,E2 386.198} C_DIS
LIN {X 35.2469,Y 76.8872,Z 89,A 60.1773,B 24.8972,C -2.3409,E1 25.0659,E2 384.569} C_DIS
LIN {X 32.9595,Y 77.8937,Z 89,A 62.018,B 24.8966,C -2.3474,E1 25.0612,E2 382.7172} C_DIS
LIN {X 30.4485,Y 78.9107,Z 89,A 63.6996,B 24.8969,C -2.3444,E1 25.0568,E2 381.0466} C_DIS
LIN {X 28.5062,Y 79.6329,Z 89,A 65.0986,B 24.8968,C -2.3455,E1 25.0532,E2 379.6478} C_DIS
LIN {X 26.5469,Y 80.3073,Z 89,A 66.7538,B 24.896,C -2.3546,E1 25.0487,E2 377.9744} C_DIS
LIN {X 23.565,Y 81.2323,Z 89,A 68.611,B 24.8965,C -2.348,E1 25.0438,E2 376.1359} C_DIS
LIN {X 21.5683,Y 81.7851,Z 89,A 70.0128,B 24.8965,C -2.3489,E1 25.04,E2 374.7343} C_DIS
LIN {X 19.5406,Y 82.2932,Z 89,A 71.4255,B 24.8965,C -2.3496,E1 25.0362,E2 373.322} C_DIS
LIN {X 17.5205,Y 82.7468,Z 89,A 72.9959,B 24.8959,C -2.3555,E1 25.0319,E2 371.7397} C_DIS
LIN {X 14.485,Y 83.3317,Z 89,A 75.1689,B 24.8956,C -2.3587,E1 25.0259,E2 369.5614} C_DIS
LIN {X 11.4044,Y 83.8089,Z 89,A 77.0312,B 24.8962,C -2.3516,E1 25.0208,E2 367.7177} C_DIS
LIN {X 9.3545,Y 84.0623,Z 89,A 78.6743,B 24.8956,C -2.3593,E1 25.0162,E2 366.0574} C_DIS
LIN {X 6.4764,Y 84.3319,Z 89,A 80.4151,B 24.8961,C -2.3528,E1 25.0114,E2 364.333} C_DIS
LIN {X 4.1919,Y 84.4772,Z 89,A 81.9378,B 24.8962,C -2.3519,E1 25.0072,E2 362.813} C_DIS
LIN {X 2.1708,Y 84.553,Z 89,A 83.308,B 24.8962,C -2.3519,E1 25.0033,E2 361.4433} C_DIS
LIN {X 0.1628,Y 84.5804,Z 89,A 84.6668,B 24.8962,C -2.3516,E1 24.9995,E2 360.0854} C_DIS
LIN {X -2.5771,Y 84.5405,Z 89,A 86.6393,B 24.896,C -2.3546,E1 24.994,E2 358.1055} C_DIS
LIN {X -5.1562,Y 84.4239,Z 89,A 88.2776,B 24.8963,C -2.3506,E1 24.9895,E2 356.4761} C_DIS
LIN {X -7.21,Y 84.2733,Z 89,A 89.674,B 24.8963,C -2.35,E1 24.9856,E2 355.0805} C_DIS
LIN {X -9.2555,Y 84.0731,Z 89,A 91.0699,B 24.8964,C -2.3494,E1 24.9817,E2 353.6853} C_DIS
LIN {X -11.3483,Y 83.8164,Z 89,A 92.4982,B 24.8965,C -2.3485,E1 24.9778,E2 352.258} C_DIS
LIN {X -13.3947,Y 83.5138,Z 89,A 93.9007,B 24.8965,C -2.3476,E1 24.9739,E2 350.8564} C_DIS
LIN {X -15.4791,Y 83.1529,Z 89,A 95.5612,B 24.8961,C -2.3533,E1 24.9693,E2 349.1808} C_DIS
LIN {X -18.4919,Y 82.535,Z 89,A 97.4242,B 24.8968,C -2.345,E1 24.9642,E2 347.3352} C_DIS
LIN {X -20.4925,Y 82.061,Z 89,A 98.8199,B 24.8969,C -2.3437,E1 24.9605,E2 345.9405} C_DIS
LIN {X -22.474,Y 81.5405,Z 89,A 100.2106,B 24.897,C -2.3424,E1 24.9567,E2 344.5509} C_DIS
LIN {X -24.2891,Y 81.0175,Z 89,A 101.5298,B 24.897,C -2.3422,E1 24.9532,E2 343.23} C_DIS
LIN {X -26.5261,Y 80.3142,Z 89,A 103.0862,B 24.8973,C -2.3394,E1 24.9491,E2 341.6774} C_DIS
LIN {X -28.4714,Y 79.6452,Z 89,A 104.4837,B 24.8975,C -2.3378,E1 24.9454,E2 340.281} C_DIS
LIN {X -30.4126,Y 78.9244,Z 89,A 105.8909,B 24.8976,C -2.3361,E1 24.9417,E2 338.875} C_DIS
LIN {X -32.348,Y 78.1511,Z 89,A 107.3035,B 24.8978,C -2.3341,E1 24.938,E2 337.4639} C_DIS
LIN {X -34.2734,Y 77.3262,Z 89,A 108.7375,B 24.8979,C -2.3325,E1 24.9344,E2 336.0304} C_DIS
LIN {X -36.1714,Y 76.4567,Z 89,A 110.1437,B 24.8981,C -2.3301,E1 24.9308,E2 334.6263} C_DIS
LIN {X -38.0332,Y 75.5479,Z 89,A 111.5544,B 24.8983,C -2.3281,E1 24.9273,E2 333.2167} C_DIS
LIN {X -39.8599,Y 74.6002,Z 89,A 112.9572,B 24.8985,C -2.326,E1 24.9238,E2 331.815} C_DIS
LIN {X -41.6752,Y 73.6014,Z 89,A 114.3662,B 24.8987,C -2.3238,E1 24.9204,E2 330.4072} C_DIS
LIN {X -43.4775,Y 72.5515,Z 89,A 115.7845,B 24.8989,C -2.3214,E1 24.917,E2 328.9904} C_DIS
LIN {X -45.2294,Y 71.4723,Z 89,A 117.1844,B 24.8991,C -2.319,E1 24.9137,E2 327.5918} C_DIS
LIN {X -46.9855,Y 70.3304,Z 89,A 118.6115,B 24.8993,C -2.3165,E1 24.9104,E2 326.1659} C_DIS
LIN {X -48.6916,Y 69.1602,Z 89,A 120.017,B 24.8996,C -2.3138,E1 24.9071,E2 324.762} C_DIS
LIN {X -50.3686,Y 67.9485,Z 89,A 121.6411,B 24.8993,C -2.3173,E1 24.9035,E2 323.1239} C_DIS
LIN {X -52.8376,Y 66.0468,Z 89,A 123.7612,B 24.8996,C -2.313,E1 24.8988,E2 321.0061} C_DIS
LIN {X -55.2174,Y 64.0704,Z 89,A 125.8756,B 24.9,C -2.3089,E1 24.8943,E2 318.8933} C_DIS
LIN {X -57.5576,Y 61.9768,Z 89,A 128.0055,B 24.9004,C -2.3041,E1 24.8899,E2 316.7663} C_DIS
LIN {X -59.7877,Y 59.8282,Z 89,A 130.1131,B 24.9008,C -2.2994,E1 24.8857,E2 314.6611} C_DIS
LIN {X -61.9347,Y 57.6026,Z 89,A 132.2145,B 24.9012,C -2.2944,E1 24.8817,E2 312.5623} C_DIS
LIN {X -64.042,Y 55.2506,Z 89,A 134.3753,B 24.9016,C -2.2896,E1 24.8777,E2 310.4033} C_DIS
LIN {X -66.023,Y 52.8673,Z 89,A 136.4843,B 24.9021,C -2.2844,E1 24.874,E2 308.2969} C_DIS
LIN {X -67.9182,Y 50.4093,Z 89,A 138.3831,B 24.9031,C -2.2732,E1 24.8709,E2 306.4158} C_DIS
LIN {X -69.1185,Y 48.7502,Z 89,A 139.7672,B 24.9034,C -2.2693,E1 24.8686,E2 305.0341} C_DIS
LIN {X -70.3193,Y 47.002,Z 89,A 141.2244,B 24.9037,C -2.2659,E1 24.8663,E2 303.5778} C_DIS
LIN {X -71.4486,Y 45.267,Z 89,A 142.6355,B 24.904,C -2.2623,E1 24.8642,E2 302.1684} C_DIS
LIN {X -72.5421,Y 43.493,Z 89,A 144.0562,B 24.9043,C -2.2585,E1 24.8621,E2 300.7494} C_DIS
LIN {X -73.5775,Y 41.7172,Z 89,A 145.4579,B 24.9046,C -2.2548,E1 24.8602,E2 299.3492} C_DIS
LIN {X -74.5703,Y 39.9154,Z 89,A 146.8621,B 24.9049,C -2.251,E1 24.8583,E2 297.9465} C_DIS
LIN {X -75.5499,Y 38.0293,Z 89,A 148.3093,B 24.9053,C -2.247,E1 24.8565,E2 296.5012} C_DIS
LIN {X -76.459,Y 36.1668,Z 89,A 149.7226,B 24.9056,C -2.2431,E1 24.8548,E2 295.0895} C_DIS
LIN {X -77.3164,Y 34.2954,Z 89,A 151.1371,B 24.9059,C -2.2395,E1 24.8532,E2 293.676} C_DIS
LIN {X -78.1464,Y 32.3595,Z 89,A 152.557,B 24.9063,C -2.235,E1 24.8516,E2 292.2589} C_DIS
LIN {X -78.9066,Y 30.4588,Z 89,A 153.959,B 24.9066,C -2.2312,E1 24.8502,E2 290.8581} C_DIS
LIN {X -79.971,Y 27.5432,Z 89,A 156.0755,B 24.9071,C -2.2251,E1 24.8482,E2 288.7441} C_DIS
LIN {X -80.6124,Y 25.6045,Z 89,A 157.4683,B 24.9075,C -2.2211,E1 24.847,E2 287.353} C_DIS
LIN {X -81.2126,Y 23.6317,Z 89,A 158.8763,B 24.9078,C -2.217,E1 24.8459,E2 285.9465} C_DIS
LIN {X -81.7879,Y 21.5582,Z 89,A 160.3431,B 24.9082,C -2.2127,E1 24.8448,E2 284.4815} C_DIS
LIN {X -82.2915,Y 19.5478,Z 89,A 161.9383,B 24.9081,C -2.2135,E1 24.8438,E2 282.8751} C_DIS
LIN {X -82.9552,Y 16.5057,Z 89,A 164.113,B 24.9085,C -2.2086,E1 24.8425,E2 280.6992} C_DIS
LIN {X -83.5072,Y 13.4371,Z 89,A 166.1871,B 24.9091,C -2.2008,E1 24.8416,E2 278.6314} C_DIS
LIN {X -83.944,Y 10.3641,Z 89,A 168.3676,B 24.9095,C -2.1963,E1 24.8408,E2 276.4487} C_DIS
LIN {X -84.2681,Y 7.2723,Z 89,A 170.2474,B 24.9106,C -2.1834,E1 24.8403,E2 274.5884} C_DIS
LIN {X -84.4798,Y 4.1436,Z 89,A 172.3847,B 24.9111,C -2.1769,E1 24.8399,E2 272.4537} C_DIS
LIN {X -84.5555,Y 2.089,Z 89,A 173.8526,B 24.9113,C -2.1745,E1 24.8399,E2 270.9827} C_DIS
LIN {X -84.5761,Y -0.8963,Z 89,A 175.8457,B 24.9119,C -2.1673,E1 24.8399,E2 268.9949} C_DIS
LIN {X -84.5245,Y -3.0986,Z 89,A 177.329,B 24.9123,C -2.1623,E1 24.8399,E2 267.5146} C_DIS
LIN {X -84.4242,Y -5.1511,Z 89,A 178.7352,B 24.9126,C -2.1582,E1 24.8401,E2 266.1096} C_DIS
LIN {X -84.2705,Y -7.2447,Z 89,A -179.8368,B 24.913,C -2.1539,E1 24.8405,E2 264.6833} C_DIS
LIN {X -84.0681,Y -9.3036,Z 89,A -178.4267,B 24.9133,C -2.1497,E1 24.8409,E2 263.2748} C_DIS
LIN {X -83.8153,Y -11.3567,Z 89,A -177.0142,B 24.9137,C -2.1456,E1 24.8414,E2 261.8636} C_DIS
LIN {X -83.5074,Y -13.4363,Z 89,A -175.3459,B 24.9135,C -2.1479,E1 24.8421,E2 260.18} C_DIS
LIN {X -82.9581,Y -16.4912,Z 89,A -173.4617,B 24.9145,C -2.1354,E1 24.8431,E2 258.3145} C_DIS
LIN {X -82.5291,Y -18.5187,Z 89,A -172.0498,B 24.9148,C -2.1313,E1 24.8439,E2 256.9041} C_DIS
LIN {X -82.0506,Y -20.535,Z 89,A -170.6363,B 24.9151,C -2.1273,E1 24.8449,E2 255.4919} C_DIS
LIN {X -81.3802,Y -23.0435,Z 89,A -168.7513,B 24.9153,C -2.1254,E1 24.8463,E2 253.6003} C_DIS
LIN {X -80.6311,Y -25.5468,Z 89,A -167.0847,B 24.9159,C -2.1173,E1 24.8476,E2 251.9436} C_DIS
LIN {X -79.9809,Y -27.5149,Z 89,A -165.6702,B 24.9162,C -2.1134,E1 24.8489,E2 250.5302} C_DIS
LIN {X -79.2826,Y -29.4665,Z 89,A -164.2483,B 24.9165,C -2.1098,E1 24.8502,E2 249.1089} C_DIS
LIN {X -78.336,Y -31.8938,Z 89,A -162.4181,B 24.9168,C -2.1065,E1 24.8521,E2 247.2762} C_DIS
LIN {X -77.3445,Y -34.2315,Z 89,A -160.7496,B 24.9173,C -2.1002,E1 24.854,E2 245.6137} C_DIS
LIN {X -76.4917,Y -36.0965,Z 89,A -159.3534,B 24.9176,C -2.0965,E1 24.8556,E2 244.2187} C_DIS
LIN {X -75.5518,Y -38.0255,Z 89,A -157.6967,B 24.9174,C -2.0981,E1 24.8577,E2 242.5491} C_DIS
LIN {X -74.0997,Y -40.7829,Z 89,A -155.7655,B 24.9183,C -2.0874,E1 24.8602,E2 240.6334} C_DIS
LIN {X -73.078,Y -42.5865,Z 89,A -154.3527,B 24.9186,C -2.0839,E1 24.8622,E2 239.2215} C_DIS
LIN {X -72.0198,Y -44.3525,Z 89,A -152.9539,B 24.9188,C -2.0804,E1 24.8642,E2 237.824} C_DIS
LIN {X -70.8965,Y -46.1269,Z 89,A -151.5211,B 24.9191,C -2.077,E1 24.8664,E2 236.3919} C_DIS
LIN {X -69.7572,Y -47.8322,Z 89,A -150.1225,B 24.9194,C -2.0738,E1 24.8686,E2 234.9942} C_DIS
LIN {X -68.579,Y -49.5064,Z 89,A -148.7286,B 24.9196,C -2.0705,E1 24.8708,E2 233.6011} C_DIS
LIN {X -67.3758,Y -51.1313,Z 89,A -147.3521,B 24.9198,C -2.0674,E1 24.8731,E2 232.2255} C_DIS
LIN {X -65.7093,Y -53.2543,Z 89,A -145.4041,B 24.9199,C -2.0665,E1 24.8765,E2 230.2705} C_DIS
LIN {X -63.699,Y -55.6433,Z 89,A -143.3875,B 24.9205,C -2.0589,E1 24.8802,E2 228.2628} C_DIS
LIN {X -61.9716,Y -57.5633,Z 89,A -141.4109,B 24.9203,C -2.0615,E1 24.8839,E2 226.2713} C_DIS
LIN {X -59.8164,Y -59.7997,Z 89,A -139.2963,B 24.9206,C -2.0573,E1 24.8881,E2 224.1576} C_DIS
LIN {X -57.5682,Y -61.967,Z 89,A -137.1695,B 24.9209,C -2.0534,E1 24.8924,E2 222.0315} C_DIS
LIN {X -55.2527,Y -64.0401,Z 89,A -135.0559,B 24.9212,C -2.0495,E1 24.8968,E2 219.9187} C_DIS
LIN {X -52.8627,Y -66.0268,Z 89,A -132.9429,B 24.9215,C -2.0459,E1 24.9014,E2 217.8064} C_DIS
LIN {X -50.3961,Y -67.9281,Z 89,A -131.0408,B 24.9223,C -2.0361,E1 24.9056,E2 215.9207} C_DIS
LIN {X -48.7057,Y -69.1503,Z 89,A -129.6193,B 24.9224,C -2.034,E1 24.9088,E2 214.4993} C_DIS
LIN {X -46.9973,Y -70.3225,Z 89,A -128.2133,B 24.9226,C -2.0319,E1 24.9121,E2 213.0937} C_DIS
LIN {X -45.2606,Y -71.4526,Z 89,A -126.8068,B 24.9227,C -2.0298,E1 24.9154,E2 211.6877} C_DIS
LIN {X -43.4847,Y -72.5472,Z 89,A -125.3902,B 24.9229,C -2.0278,E1 24.9188,E2 210.2714} C_DIS
LIN {X -40.7899,Y -74.0958,Z 89,A -123.2779,B 24.9231,C -2.0251,E1 24.9239,E2 208.1594} C_DIS
LIN {X -38.9577,Y -75.0753,Z 89,A -121.8662,B 24.9232,C -2.0234,E1 24.9274,E2 206.7478} C_DIS
LIN {X -37.1248,Y -75.9983,Z 89,A -120.3257,B 24.923,C -2.0262,E1 24.9313,E2 205.1966} C_DIS
LIN {X -34.4587,Y -77.2428,Z 89,A -118.4503,B 24.9235,C -2.0205,E1 24.936,E2 203.3301} C_DIS
LIN {X -32.3645,Y -78.1444,Z 89,A -116.9282,B 24.9236,C -2.0182,E1 24.9399,E2 201.81} C_DIS
LIN {X -30.4534,Y -78.9087,Z 89,A -115.5288,B 24.9237,C -2.017,E1 24.9436,E2 200.4103} C_DIS
LIN {X -27.9314,Y -79.8347,Z 89,A -113.6251,B 24.9237,C -2.018,E1 24.9486,E2 198.5006} C_DIS
LIN {X -25.5662,Y -80.6248,Z 89,A -112.0133,B 24.9239,C -2.0143,E1 24.9528,E2 196.8945} C_DIS
LIN {X -23.5704,Y -81.2308,Z 89,A -110.598,B 24.9239,C -2.0134,E1 24.9566,E2 195.479} C_DIS
LIN {X -21.5567,Y -81.7883,Z 89,A -109.1807,B 24.924,C -2.0126,E1 24.9605,E2 194.0615} C_DIS
LIN {X -19.5488,Y -82.2913,Z 89,A -107.7767,B 24.9241,C -2.0119,E1 24.9643,E2 192.6572} C_DIS
LIN {X -17.5293,Y -82.7449,Z 89,A -106.1353,B 24.9236,C -2.0186,E1 24.9688,E2 190.9979} C_DIS
LIN {X -14.4833,Y -83.332,Z 89,A -104.2701,B 24.9242,C -2.0106,E1 24.9739,E2 189.1497} C_DIS
LIN {X -12.4473,Y -83.6603,Z 89,A -102.8726,B 24.9242,C -2.0103,E1 24.9777,E2 187.7518} C_DIS
LIN {X -9.7822,Y -84.0122,Z 89,A -100.9598,B 24.924,C -2.0128,E1 24.9831,E2 185.8316} C_DIS
LIN {X -7.271,Y -84.2682,Z 89,A -99.3407,B 24.9243,C -2.0099,E1 24.9875,E2 184.2187} C_DIS
LIN {X -4.9637,Y -84.4346,Z 89,A -97.8122,B 24.9243,C -2.0087,E1 24.9918,E2 182.6924} C_DIS
LIN {X -3.0153,Y -84.5271,Z 89,A -96.4828,B 24.9243,C -2.0091,E1 24.9955,E2 181.3618} C_DIS
LIN {X -1.0103,Y -84.5752,Z 89,A -95.1115,B 24.9243,C -2.0097,E1 24.9993,E2 179.9889} C_DIS
LIN {X -1.0103,Y -84.5752,Z 89,A -95.1115,B 24.9243,C -2.0097,E1 24.9993,E2 179.9889} C_DIS
Enddeposition()
LIN {X 0.6173,Y -92.6509,Z 90,A -94.2891,B 24.9346,C -1.8679,E1 25.0007,E2 179.5031} C_DIS
Startdeposition()
$VEL.CP = VEL_PRINT
LIN {X 2.9017,Y -92.6095,Z 90,A -92.2333,B 24.933,C -1.8904,E1 25.0066,E2 177.3941} C_DIS
LIN {X 6.1896,Y -92.4479,Z 90,A -90.1617,B 24.9329,C -1.8925,E1 25.0124,E2 175.3183} C_DIS
LIN {X 9.5882,Y -92.1575,Z 90,A -88.0548,B 24.9328,C -1.8936,E1 25.0182,E2 173.2102} C_DIS
LIN {X 12.9737,Y -91.7421,Z 90,A -85.9485,B 24.9327,C -1.8948,E1 25.0241,E2 171.1027} C_DIS
LIN {X 16.4589,Y -91.1813,Z 90,A -83.8067,B 24.9327,C -1.895,E1 25.03,E2 168.9626} C_DIS
LIN {X 19.8039,Y -90.5137,Z 90,A -81.7013,B 24.9326,C -1.8968,E1 25.0357,E2 166.8558} C_DIS
LIN {X 23.0067,Y -89.7531,Z 90,A -79.6324,B 24.9323,C -1.9,E1 25.0413,E2 164.7824} C_DIS
LIN {X 26.2947,Y -88.8455,Z 90,A -77.528,B 24.9322,C -1.9021,E1 25.047,E2 162.6763} C_DIS
LIN {X 29.6598,Y -87.7794,Z 90,A -75.3886,B 24.9321,C -1.9032,E1 25.0527,E2 160.5384} C_DIS
LIN {X 32.7593,Y -86.6704,Z 90,A -73.3212,B 24.9318,C -1.907,E1 25.0581,E2 158.4663} C_DIS
LIN {X 35.9272,Y -85.4059,Z 90,A -71.2184,B 24.9316,C -1.9098,E1 25.0635,E2 156.3617} C_DIS
LIN {X 39.1543,Y -83.9754,Z 90,A -69.0804,B 24.9315,C -1.9115,E1 25.069,E2 154.225} C_DIS
LIN {X 42.2187,Y -82.4773,Z 90,A -66.9785,B 24.9313,C -1.9147,E1 25.0742,E2 152.1212} C_DIS
LIN {X 45.2259,Y -80.8675,Z 90,A -64.8771,B 24.931,C -1.9181,E1 25.0794,E2 150.0179} C_DIS
LIN {X 48.07,Y -79.2099,Z 90,A -62.8119,B 24.9307,C -1.9229,E1 25.0844,E2 147.9477} C_DIS
LIN {X 50.9529,Y -77.3869,Z 90,A -60.7115,B 24.9304,C -1.9267,E1 25.0893,E2 145.8453} C_DIS
LIN {X 53.8637,Y -75.3899,Z 90,A -58.5757,B 24.9302,C -1.9294,E1 25.0942,E2 143.7105} C_DIS
LIN {X 56.5078,Y -73.4289,Z 90,A -56.5117,B 24.9298,C -1.9347,E1 25.0988,E2 141.6413} C_DIS
LIN {X 59.1722,Y -71.2992,Z 90,A -54.4126,B 24.9295,C -1.939,E1 25.1033,E2 139.5401} C_DIS
LIN {X 61.7565,Y -69.0729,Z 90,A -52.3137,B 24.9292,C -1.9434,E1 25.1077,E2 137.439} C_DIS
LIN {X 64.3427,Y -66.6704,Z 90,A -50.1797,B 24.9289,C -1.9468,E1 25.1121,E2 135.3058} C_DIS
LIN {X 66.6704,Y -64.3427,Z 90,A -48.1172,B 24.9285,C -1.9528,E1 25.1161,E2 133.2379} C_DIS
LIN {X 69.0729,Y -61.7565,Z 90,A -45.9838,B 24.9282,C -1.9564,E1 25.1201,E2 131.1053} C_DIS
LIN {X 71.2992,Y -59.1722,Z 90,A -43.8863,B 24.9279,C -1.9615,E1 25.1239,E2 129.0055} C_DIS
LIN {X 73.4289,Y -56.5078,Z 90,A -41.7891,B 24.9275,C -1.9666,E1 25.1276,E2 126.9059} C_DIS
LIN {X 75.3899,Y -53.8637,Z 90,A -39.7279,B 24.927,C -1.9731,E1 25.1309,E2 124.8394} C_DIS
LIN {X 77.3869,Y -50.9529,Z 90,A -37.5958,B 24.9267,C -1.9773,E1 25.1343,E2 122.7079} C_DIS
LIN {X 79.2099,Y -48.07,Z 90,A -35.4994,B 24.9263,C -1.9828,E1 25.1374,E2 120.6091} C_DIS
LIN {X 80.8675,Y -45.2259,Z 90,A -33.439,B 24.9258,C -1.9897,E1 25.1402,E2 118.5433} C_DIS
LIN {X 82.4773,Y -42.2187,Z 90,A -31.3433,B 24.9253,C -1.9954,E1 25.1429,E2 116.4451} C_DIS
LIN {X 83.9754,Y -39.1543,Z 90,A -29.2476,B 24.9249,C -2.0012,E1 25.1455,E2 114.3471} C_DIS
LIN {X 85.4059,Y -35.9272,Z 90,A -27.1166,B 24.9246,C -2.0058,E1 25.1478,E2 112.2167} C_DIS
LIN {X 86.6704,Y -32.7593,Z 90,A -25.0213,B 24.9241,C -2.0118,E1 25.15,E2 110.119} C_DIS
LIN {X 87.7794,Y -29.6598,Z 90,A -22.9616,B 24.9236,C -2.019,E1 25.1519,E2 108.0539} C_DIS
LIN {X 88.8455,Y -26.2947,Z 90,A -20.8312,B 24.9232,C -2.0239,E1 25.1536,E2 105.9241} C_DIS
LIN {X 89.7531,Y -23.0067,Z 90,A -18.7362,B 24.9227,C -2.03,E1 25.1551,E2 103.8267} C_DIS
LIN {X 90.5137,Y -19.8039,Z 90,A -16.677,B 24.9222,C -2.0373,E1 25.1564,E2 101.7621} C_DIS
LIN {X 91.1813,Y -16.4589,Z 90,A -14.5825,B 24.9217,C -2.0435,E1 25.1575,E2 99.6652} C_DIS
LIN {X 91.7421,Y -12.9737,Z 90,A -12.4523,B 24.9213,C -2.0485,E1 25.1584,E2 97.5358} C_DIS
LIN {X 92.1575,Y -9.5882,Z 90,A -10.3575,B 24.9208,C -2.0548,E1 25.1591,E2 95.4387} C_DIS
LIN {X 92.4479,Y -6.1896,Z 90,A -8.263,B 24.9203,C -2.061,E1 25.1595,E2 93.342} C_DIS
LIN {X 92.6095,Y -2.9017,Z 90,A -6.204,B 24.9198,C -2.0684,E1 25.1597,E2 91.2776} C_DIS
LIN {X 92.6576,Y 0.0827,Z 90,A -4.2839,B 24.9191,C -2.0771,E1 25.1597,E2 89.3485} C_DIS
LIN {X 92.5938,Y 3.4104,Z 90,A -2.2544,B 24.9187,C -2.0826,E1 25.1597,E2 87.3181} C_DIS
LIN {X 92.4056,Y 6.8162,Z 90,A -0.1296,B 24.9181,C -2.0899,E1 25.1592,E2 85.1886} C_DIS
LIN {X 92.0921,Y 10.2128,Z 90,A 1.9652,B 24.9176,C -2.096,E1 25.1586,E2 83.0917} C_DIS
LIN {X 91.6537,Y 13.5955,Z 90,A 4.03,B 24.9172,C -2.101,E1 25.1578,E2 81.0275} C_DIS
LIN {X 91.0912,Y 16.9599,Z 90,A 6.125,B 24.9167,C -2.107,E1 25.1568,E2 78.9304} C_DIS
LIN {X 90.4053,Y 20.3012,Z 90,A 8.2502,B 24.9162,C -2.1142,E1 25.1555,E2 76.8008} C_DIS
LIN {X 89.5968,Y 23.615,Z 90,A 10.3154,B 24.9158,C -2.1189,E1 25.1541,E2 74.7362} C_DIS
LIN {X 88.6669,Y 26.8968,Z 90,A 12.441,B 24.9152,C -2.1259,E1 25.1524,E2 72.6063} C_DIS
LIN {X 87.6168,Y 30.1421,Z 90,A 14.5366,B 24.9148,C -2.1317,E1 25.1506,E2 70.5089} C_DIS
LIN {X 86.448,Y 33.3467,Z 90,A 16.6327,B 24.9143,C -2.1374,E1 25.1485,E2 68.4111} C_DIS
LIN {X 85.162,Y 36.506,Z 90,A 18.7287,B 24.9139,C -2.1429,E1 25.1462,E2 66.3135} C_DIS
LIN {X 83.7606,Y 39.6158,Z 90,A 20.8252,B 24.9134,C -2.1484,E1 25.1438,E2 64.2153} C_DIS
LIN {X 82.2457,Y 42.672,Z 90,A 22.8918,B 24.9131,C -2.1526,E1 25.1411,E2 62.1497} C_DIS
LIN {X 80.6193,Y 45.6703,Z 90,A 24.9888,B 24.9127,C -2.1579,E1 25.1383,E2 60.0513} C_DIS
LIN {X 78.8837,Y 48.6067,Z 90,A 27.116,B 24.9122,C -2.1641,E1 25.1352,E2 57.9203} C_DIS
LIN {X 77.0412,Y 51.4773,Z 90,A 29.1834,B 24.9118,C -2.168,E1 25.132,E2 55.854} C_DIS
LIN {X 75.0942,Y 54.278,Z 90,A 31.2813,B 24.9114,C -2.1728,E1 25.1287,E2 53.7549} C_DIS
LIN {X 73.0455,Y 57.0053,Z 90,A 33.4098,B 24.911,C -2.1786,E1 25.125,E2 51.6228} C_DIS
LIN {X 70.8978,Y 59.6553,Z 90,A 35.478,B 24.9107,C -2.1821,E1 25.1213,E2 49.556} C_DIS
LIN {X 68.654,Y 62.2244,Z 90,A 37.577,B 24.9103,C -2.1864,E1 25.1174,E2 47.456} C_DIS
LIN {X 66.3172,Y 64.7092,Z 90,A 39.6765,B 24.91,C -2.1907,E1 25.1134,E2 45.3556} C_DIS
LIN {X 63.8905,Y 67.1063,Z 90,A 41.8065,B 24.9096,C -2.1958,E1 25.1091,E2 43.2223} C_DIS
LIN {X 61.3772,Y 69.4124,Z 90,A 43.9066,B 24.9092,C -2.1997,E1 25.1047,E2 41.1215} C_DIS
LIN {X 58.7807,Y 71.6245,Z 90,A 45.9771,B 24.909,C -2.2023,E1 25.1003,E2 39.0527} C_DIS
LIN {X 56.1046,Y 73.7396,Z 90,A 48.078,B 24.9087,C -2.2058,E1 25.0957,E2 36.9513} C_DIS
LIN {X 53.3524,Y 75.7546,Z 90,A 50.1796,B 24.9085,C -2.2091,E1 25.0909,E2 34.8492} C_DIS
LIN {X 50.528,Y 77.6671,Z 90,A 52.2815,B 24.9082,C -2.2122,E1 25.086,E2 32.7469} C_DIS
LIN {X 47.635,Y 79.4742,Z 90,A 54.384,B 24.908,C -2.2151,E1 25.081,E2 30.6441} C_DIS
LIN {X 44.6775,Y 81.1737,Z 90,A 56.4869,B 24.9077,C -2.2178,E1 25.0759,E2 28.541} C_DIS
LIN {X 41.6595,Y 82.7631,Z 90,A 58.5904,B 24.9075,C -2.2204,E1 25.0706,E2 26.4373} C_DIS
LIN {X 38.585,Y 84.2404,Z 90,A 60.6943,B 24.9073,C -2.2227,E1 25.0653,E2 24.3334} C_DIS
LIN {X 35.4582,Y 85.6036,Z 90,A 62.829,B 24.9071,C -2.2258,E1 25.0598,E2 22.1963} C_DIS
LIN {X 32.2833,Y 86.8507,Z 90,A 64.9036,B 24.907,C -2.2266,E1 25.0544,E2 20.1243} C_DIS
LIN {X 29.0647,Y 87.9801,Z 90,A 67.0092,B 24.9069,C -2.2282,E1 25.0488,E2 18.0189} C_DIS
LIN {X 25.8067,Y 88.9902,Z 90,A 69.1151,B 24.9067,C -2.2297,E1 25.0432,E2 15.9133} C_DIS
LIN {X 22.5137,Y 89.8798,Z 90,A 71.2217,B 24.9067,C -2.2309,E1 25.0375,E2 13.8071} C_DIS
LIN {X 19.1902,Y 90.6476,Z 90,A 73.3287,B 24.9066,C -2.2318,E1 25.0318,E2 11.7005} C_DIS
LIN {X 15.8408,Y 91.2925,Z 90,A 75.4364,B 24.9065,C -2.2326,E1 25.026,E2 9.5934} C_DIS
LIN {X 12.4698,Y 91.8137,Z 90,A 77.5445,B 24.9065,C -2.2331,E1 25.0202,E2 7.486} C_DIS
LIN {X 9.0819,Y 92.2105,Z 90,A 79.6532,B 24.9065,C -2.2334,E1 25.0143,E2 5.3781} C_DIS
LIN {X 5.6818,Y 92.4822,Z 90,A 81.7927,B 24.9063,C -2.2345,E1 25.0083,E2 3.237} C_DIS
LIN {X 2.2739,Y 92.6287,Z 90,A 83.9026,B 24.9063,C -2.2343,E1 25.0025,E2 1.1279} C_DIS
LIN {X -1.137,Y 92.6496,Z 90,A 86.0128,B 24.9063,C -2.2339,E1 24.9966,E2 -0.9813} C_DIS
LIN {X -4.5464,Y 92.545,Z 90,A 88.0934,B 24.9065,C -2.2322,E1 24.9908,E2 -3.0584} C_DIS
LIN {X -7.9497,Y 92.315,Z 90,A 90.2047,B 24.9065,C -2.2314,E1 24.9849,E2 -5.1686} C_DIS
LIN {X -11.3422,Y 91.9598,Z 90,A 92.3471,B 24.9066,C -2.2313,E1 24.9789,E2 -7.3121} C_DIS
LIN {X -14.7193,Y 91.48,Z 90,A 94.4597,B 24.9067,C -2.23,E1 24.9731,E2 -9.4234} C_DIS
LIN {X -18.0764,Y 90.8762,Z 90,A 96.5726,B 24.9068,C -2.2284,E1 24.9673,E2 -11.5349} C_DIS
LIN {X -21.4091,Y 90.1493,Z 90,A 98.6558,B 24.9071,C -2.2256,E1 24.9617,E2 -13.6142} C_DIS
LIN {X -24.7127,Y 89.3002,Z 90,A 100.77,B 24.9072,C -2.2237,E1 24.956,E2 -15.7269} C_DIS
LIN {X -27.9828,Y 88.3301,Z 90,A 102.9149,B 24.9073,C -2.2224,E1 24.9502,E2 -17.8726} C_DIS
LIN {X -31.2151,Y 87.2403,Z 90,A 104.9997,B 24.9076,C -2.219,E1 24.9448,E2 -19.9534} C_DIS
LIN {X -34.405,Y 86.0322,Z 90,A 107.1154,B 24.9079,C -2.2164,E1 24.9393,E2 -22.0673} C_DIS
LIN {X -37.5483,Y 84.7076,Z 90,A 109.2619,B 24.908,C -2.2145,E1 24.9338,E2 -24.2145} C_DIS
LIN {X -40.6407,Y 83.2681,Z 90,A 111.3786,B 24.9083,C -2.2115,E1 24.9284,E2 -26.3294} C_DIS
LIN {X -43.678,Y 81.7158,Z 90,A 113.4652,B 24.9086,C -2.2073,E1 24.9233,E2 -28.4117} C_DIS
LIN {X -46.6562,Y 80.0528,Z 90,A 115.5827,B 24.9089,C -2.2038,E1 24.9182,E2 -30.5271} C_DIS
LIN {X -49.5711,Y 78.2813,Z 90,A 117.7008,B 24.9092,C -2.2002,E1 24.9131,E2 -32.6433} C_DIS
LIN {X -52.4188,Y 76.4037,Z 90,A 119.8496,B 24.9094,C -2.1973,E1 24.9082,E2 -34.7925} C_DIS
LIN {X -55.1955,Y 74.4225,Z 90,A 121.9381,B 24.9098,C -2.1923,E1 24.9035,E2 -36.8765} C_DIS
LIN {X -57.8974,Y 72.3405,Z 90,A 124.0574,B 24.9102,C -2.1882,E1 24.8988,E2 -38.9936} C_DIS
LIN {X -60.5208,Y 70.1604,Z 90,A 126.2077,B 24.9105,C -2.1848,E1 24.8942,E2 -41.1442} C_DIS
LIN {X -63.0622,Y 67.8853,Z 90,A 128.3278,B 24.9108,C -2.1802,E1 24.8899,E2 -43.262} C_DIS
LIN {X -65.5181,Y 65.5181,Z 90,A 130.4177,B 24.9113,C -2.1746,E1 24.8857,E2 -45.3473} C_DIS
LIN {X -67.8853,Y 63.0622,Z 90,A 132.5691,B 24.9116,C -2.1707,E1 24.8816,E2 -47.4987} C_DIS
LIN {X -70.1604,Y 60.5208,Z 90,A 134.6598,B 24.9121,C -2.1648,E1 24.8778,E2 -49.5848} C_DIS
LIN {X -72.3405,Y 57.8974,Z 90,A 136.8118,B 24.9124,C -2.1606,E1 24.874,E2 -51.7369} C_DIS
LIN {X -74.4225,Y 55.1955,Z 90,A 138.9031,B 24.9129,C -2.1544,E1 24.8705,E2 -53.8234} C_DIS
LIN {X -76.4037,Y 52.4188,Z 90,A 141.0559,B 24.9133,C -2.15,E1 24.867,E2 -55.9761} C_DIS
LIN {X -78.2813,Y 49.5711,Z 90,A 143.1782,B 24.9137,C -2.1445,E1 24.8638,E2 -58.0961} C_DIS
LIN {X -80.0528,Y 46.6562,Z 90,A 145.3009,B 24.9142,C -2.1389,E1 24.8608,E2 -60.2164} C_DIS
LIN {X -81.7158,Y 43.678,Z 90,A 147.4237,B 24.9147,C -2.1332,E1 24.858,E2 -62.3368} C_DIS
LIN {X -83.2681,Y 40.6407,Z 90,A 149.5471,B 24.9151,C -2.1274,E1 24.8553,E2 -64.4577} C_DIS
LIN {X -84.7076,Y 37.5483,Z 90,A 151.6703,B 24.9156,C -2.1215,E1 24.8529,E2 -66.5786} C_DIS
LIN {X -86.0322,Y 34.405,Z 90,A 153.7938,B 24.9161,C -2.1155,E1 24.8506,E2 -68.6996} C_DIS
LIN {X -87.2403,Y 31.2151,Z 90,A 155.8872,B 24.9166,C -2.1085,E1 24.8486,E2 -70.7882} C_DIS
LIN {X -88.3301,Y 27.9828,Z 90,A 158.0414,B 24.917,C -2.1034,E1 24.8468,E2 -72.9424} C_DIS
LIN {X -89.3002,Y 24.7127,Z 90,A 160.1654,B 24.9175,C -2.0972,E1 24.8452,E2 -75.064} C_DIS
LIN {X -90.1493,Y 21.4091,Z 90,A 162.2588,B 24.9181,C -2.0901,E1 24.8438,E2 -77.1526} C_DIS
LIN {X -90.8762,Y 18.0764,Z 90,A 164.3831,B 24.9186,C -2.0838,E1 24.8426,E2 -79.2745} C_DIS
LIN {X -91.48,Y 14.7193,Z 90,A 166.5074,B 24.9191,C -2.0776,E1 24.8416,E2 -81.3965} C_DIS
LIN {X -91.9598,Y 11.3422,Z 90,A 168.6622,B 24.9195,C -2.0722,E1 24.8408,E2 -83.5514} C_DIS
LIN {X -92.315,Y 7.9497,Z 90,A 170.7866,B 24.92,C -2.0659,E1 24.8402,E2 -85.6735} C_DIS
LIN {X -92.545,Y 4.5464,Z 90,A 172.8804,B 24.9205,C -2.0587,E1 24.8399,E2 -87.7626} C_DIS
LIN {X -92.6496,Y 1.137,Z 90,A 174.7803,B 24.9215,C -2.0455,E1 24.8398,E2 -89.6425} C_DIS
LIN {X -92.6403,Y -1.646,Z 90,A 176.664,B 24.9215,C -2.045,E1 24.8398,E2 -91.5364} C_DIS
LIN {X -92.5169,Y -5.0547,Z 90,A 178.7882,B 24.9221,C -2.0387,E1 24.8401,E2 -93.6584} C_DIS
LIN {X -92.2572,Y -8.5751,Z 90,A -179.0518,B 24.9226,C -2.0311,E1 24.8406,E2 -95.8132} C_DIS
LIN {X -91.8791,Y -11.965,Z 90,A -176.9274,B 24.9231,C -2.0249,E1 24.8413,E2 -97.9356} C_DIS
LIN {X -91.3961,Y -15.2213,Z 90,A -174.8397,B 24.9235,C -2.0202,E1 24.8422,E2 -100.0243} C_DIS
LIN {X -90.7739,Y -18.575,Z 90,A -172.7156,B 24.9239,C -2.0141,E1 24.8433,E2 -102.1464} C_DIS
LIN {X -90.0287,Y -21.9036,Z 90,A -170.5921,B 24.9244,C -2.008,E1 24.8447,E2 -104.268} C_DIS
LIN {X -89.1615,Y -25.2024,Z 90,A -168.4684,B 24.9248,C -2.0021,E1 24.8462,E2 -106.3898} C_DIS
LIN {X -88.1734,Y -28.4671,Z 90,A -166.3431,B 24.9253,C -1.9963,E1 24.848,E2 -108.5135} C_DIS
LIN {X -87.0251,Y -31.8051,Z 90,A -164.1863,B 24.9258,C -1.989,E1 24.85,E2 -110.6653} C_DIS
LIN {X -85.7955,Y -34.9867,Z 90,A -162.0632,B 24.9262,C -1.9834,E1 24.8522,E2 -112.7867} C_DIS
LIN {X -84.4496,Y -38.1209,Z 90,A -159.9406,B 24.9267,C -1.9778,E1 24.8546,E2 -114.9076} C_DIS
LIN {X -82.9892,Y -41.2034,Z 90,A -157.818,B 24.9271,C -1.9723,E1 24.8572,E2 -117.0287} C_DIS
LIN {X -81.4164,Y -44.2301,Z 90,A -155.6962,B 24.9275,C -1.967,E1 24.8599,E2 -119.149} C_DIS
LIN {X -79.7938,Y -47.0944,Z 90,A -153.6104,B 24.9277,C -1.9631,E1 24.8628,E2 -121.2365} C_DIS
LIN {X -78.0063,Y -49.9994,Z 90,A -151.489,B 24.9281,C -1.958,E1 24.866,E2 -123.3566} C_DIS
LIN {X -76.0452,Y -52.9345,Z 90,A -149.3318,B 24.9286,C -1.9517,E1 24.8694,E2 -125.5093} C_DIS
LIN {X -74.1168,Y -55.6025,Z 90,A -147.2471,B 24.9288,C -1.9483,E1 24.8728,E2 -127.5959} C_DIS
LIN {X -72.02,Y -58.2928,Z 90,A -145.1267,B 24.9292,C -1.9436,E1 24.8765,E2 -129.7152} C_DIS
LIN {X -69.8256,Y -60.9042,Z 90,A -143.0065,B 24.9295,C -1.9391,E1 24.8804,E2 -131.8345} C_DIS
LIN {X -67.5366,Y -63.433,Z 90,A -140.887,B 24.9298,C -1.9348,E1 24.8844,E2 -133.953} C_DIS
LIN {X -65.0713,Y -65.9595,Z 90,A -138.7319,B 24.9302,C -1.9293,E1 24.8886,E2 -136.1042} C_DIS
LIN {X -62.5994,Y -68.3099,Z 90,A -136.6094,B 24.9305,C -1.9255,E1 24.8929,E2 -138.2262} C_DIS
LIN {X -60.1333,Y -70.4905,Z 90,A -134.5306,B 24.9307,C -1.9229,E1 24.8973,E2 -140.307} C_DIS
LIN {X -57.498,Y -72.6561,Z 90,A -132.4127,B 24.9309,C -1.9193,E1 24.9019,E2 -142.4243} C_DIS
LIN {X -54.7848,Y -74.7232,Z 90,A -130.2954,B 24.9312,C -1.9159,E1 24.9066,E2 -144.5411} C_DIS
LIN {X -51.9973,Y -76.689,Z 90,A -128.1784,B 24.9314,C -1.9127,E1 24.9115,E2 -146.6577} C_DIS
LIN {X -49.0384,Y -78.614,Z 90,A -126.0261,B 24.9317,C -1.9084,E1 24.9166,E2 -148.8065} C_DIS
LIN {X -46.2148,Y -80.3064,Z 90,A -123.9458,B 24.9318,C -1.9069,E1 24.9216,E2 -150.8897} C_DIS
LIN {X -43.1223,Y -82.0085,Z 90,A -121.7944,B 24.9321,C -1.903,E1 24.9269,E2 -153.0377} C_DIS
LIN {X -40.1819,Y -83.4886,Z 90,A -119.7154,B 24.9321,C -1.902,E1 24.9321,E2 -155.1198} C_DIS
LIN {X -37.0817,Y -84.911,Z 90,A -117.6009,B 24.9323,C -1.8998,E1 24.9375,E2 -157.2343} C_DIS
LIN {X -33.9312,Y -86.2183,Z 90,A -115.4869,B 24.9325,C -1.8979,E1 24.9429,E2 -159.3483} C_DIS
LIN {X -30.7348,Y -87.4088,Z 90,A -113.3735,B 24.9325,C -1.8962,E1 24.9485,E2 -161.4619} C_DIS
LIN {X -27.4967,Y -88.4809,Z 90,A -111.2607,B 24.9327,C -1.8947,E1 24.9541,E2 -163.575} C_DIS
LIN {X -24.2213,Y -89.433,Z 90,A -109.1481,B 24.9327,C -1.8934,E1 24.9598,E2 -165.688} C_DIS
LIN {X -20.7971,Y -90.2907,Z 90,A -107.0006,B 24.933,C -1.8911,E1 24.9656,E2 -167.8328} C_DIS
LIN {X -17.5766,Y -90.9725,Z 90,A -104.9251,B 24.933,C -1.8916,E1 24.9713,E2 -169.9119} C_DIS
LIN {X -14.2162,Y -91.5578,Z 90,A -102.8145,B 24.933,C -1.891,E1 24.9771,E2 -172.0232} C_DIS
LIN {X -10.8366,Y -92.019,Z 90,A -100.7042,B 24.933,C -1.8907,E1 24.983,E2 -174.1342} C_DIS
LIN {X -7.4423,Y -92.3555,Z 90,A -98.5946,B 24.933,C -1.8906,E1 24.9888,E2 -176.2446} C_DIS
LIN {X -3.919,Y -92.572,Z 90,A -96.4498,B 24.933,C -1.8894,E1 24.9948,E2 -178.3871} C_DIS
LIN {X -0.509,Y -92.6535,Z 90,A -94.3412,B 24.933,C -1.8898,E1 25.0007,E2 -180.4967} C_DIS
LIN {X -0.509,Y -92.6535,Z 90,A -94.3412,B 24.933,C -1.8898,E1 25.0007,E2 -180.4967} C_DIS
Enddeposition()
LIN {X 0.6231,Y -91.6697,Z 90,A -94.7607,B 24.9345,C -1.869,E1 24.9994,E2 -180.028} C_DIS
Startdeposition()
$VEL.CP = VEL_PRINT
LIN {X -6.4519,Y -91.4474,Z 90,A -99.0264,B 24.9342,C -1.8738,E1 24.9875,E2 -175.7728} C_DIS
LIN {X -10.1022,Y -91.1178,Z 90,A -101.3089,B 24.9342,C -1.8743,E1 24.9812,E2 -173.4901} C_DIS
LIN {X -13.9172,Y -90.6119,Z 90,A -103.8362,B 24.9344,C -1.8708,E1 24.9742,E2 -170.9525} C_DIS
LIN {X -17.5906,Y -89.9712,Z 90,A -106.0648,B 24.9341,C -1.875,E1 24.9681,E2 -168.7315} C_DIS
LIN {X -21.1625,Y -89.1999,Z 90,A -108.2903,B 24.9339,C -1.878,E1 24.962,E2 -166.5103} C_DIS
LIN {X -24.0987,Y -88.4504,Z 90,A -110.2724,B 24.934,C -1.8762,E1 24.9566,E2 -164.5211} C_DIS
LIN {X -27.2764,Y -87.5226,Z 90,A -112.3124,B 24.9338,C -1.8787,E1 24.9512,E2 -162.4833} C_DIS
LIN {X -31.1958,Y -86.2036,Z 90,A -114.9045,B 24.9338,C -1.8806,E1 24.9444,E2 -159.8908} C_DIS
LIN {X -34.7731,Y -84.8237,Z 90,A -117.2887,B 24.9335,C -1.8833,E1 24.9382,E2 -157.5079} C_DIS
LIN {X -38.0448,Y -83.4084,Z 90,A -119.8877,B 24.9342,C -1.8738,E1 24.9315,E2 -154.8801} C_DIS
LIN {X -42.0146,Y -81.4805,Z 90,A -122.148,B 24.9328,C -1.8931,E1 24.9259,E2 -152.6597} C_DIS
LIN {X -45.0696,Y -79.8317,Z 90,A -124.2879,B 24.9325,C -1.897,E1 24.9207,E2 -150.5229} C_DIS
LIN {X -47.4176,Y -78.459,Z 90,A -126.1361,B 24.9327,C -1.8947,E1 24.9162,E2 -148.6637} C_DIS
LIN {X -50.2578,Y -76.6707,Z 90,A -128.2891,B 24.9326,C -1.8962,E1 24.9112,E2 -146.5072} C_DIS
LIN {X -54.5056,Y -73.7124,Z 90,A -131.6014,B 24.9324,C -1.8992,E1 24.9036,E2 -143.1906} C_DIS
LIN {X -57.1824,Y -71.6558,Z 90,A -133.7547,B 24.9322,C -1.9016,E1 24.8989,E2 -141.0351} C_DIS
LIN {X -60.1488,Y -69.1835,Z 90,A -136.0441,B 24.9316,C -1.9101,E1 24.894,E2 -138.757} C_DIS
LIN {X -62.7766,Y -66.8078,Z 90,A -138.5841,B 24.932,C -1.9044,E1 24.8888,E2 -136.1932} C_DIS
LIN {X -66.2441,Y -63.3721,Z 90,A -141.4208,B 24.9311,C -1.9175,E1 24.8833,E2 -133.3755} C_DIS
LIN {X -68.7228,Y -60.6763,Z 90,A -143.983,B 24.9313,C -1.9142,E1 24.8785,E2 -130.794} C_DIS
LIN {X -70.9522,Y -58.053,Z 90,A -145.8627,B 24.9303,C -1.9275,E1 24.8751,E2 -128.9374} C_DIS
LIN {X -73.0346,Y -55.4106,Z 90,A -147.9486,B 24.9299,C -1.9331,E1 24.8716,E2 -126.8549} C_DIS
LIN {X -75.928,Y -51.3725,Z 90,A -150.9626,B 24.9292,C -1.9436,E1 24.8668,E2 -123.8511} C_DIS
LIN {X -77.6448,Y -48.7392,Z 90,A -153.0356,B 24.929,C -1.9454,E1 24.8636,E2 -121.7719} C_DIS
LIN {X -80.1688,Y -44.4659,Z 90,A -157.3201,B 24.931,C -1.9182,E1 24.8576,E2 -117.4002} C_DIS
LIN {X -82.7988,Y -39.3536,Z 90,A -159.5626,B 24.9273,C -1.9686,E1 24.855,E2 -115.2657} C_DIS
LIN {X -83.7569,Y -37.2715,Z 90,A -161.2793,B 24.9277,C -1.964,E1 24.853,E2 -113.5288} C_DIS
LIN {X -85.0455,Y -34.2283,Z 90,A -163.2303,B 24.927,C -1.9734,E1 24.8509,E2 -111.5893} C_DIS
LIN {X -86.1075,Y -31.4593,Z 90,A -165.0799,B 24.9266,C -1.979,E1 24.8491,E2 -109.7426} C_DIS
LIN {X -87.317,Y -27.9289,Z 90,A -168.0351,B 24.9274,C -1.9673,E1 24.8465,E2 -106.7426} C_DIS
LIN {X -88.3526,Y -24.4603,Z 90,A -169.7181,B 24.9256,C -1.9914,E1 24.8453,E2 -105.1073} C_DIS
LIN {X -89.2215,Y -21.069,Z 90,A -172.0018,B 24.9254,C -1.9952,E1 24.8437,E2 -102.8193} C_DIS
LIN {X -89.8777,Y -18.0648,Z 90,A -173.9545,B 24.925,C -2.0002,E1 24.8426,E2 -100.8671} C_DIS
LIN {X -90.5166,Y -14.5317,Z 90,A -176.1711,B 24.9244,C -2.008,E1 24.8416,E2 -98.656} C_DIS
LIN {X -90.9335,Y -11.6324,Z 90,A -178.0471,B 24.9241,C -2.0124,E1 24.8409,E2 -96.7793} C_DIS
LIN {X -91.3289,Y -7.9643,Z 90,A 179.5922,B 24.9236,C -2.0181,E1 24.8403,E2 -94.418} C_DIS
Enddeposition()
END
